  MoveL (T18222) to (121.46, 121.46, 19.3) mm, rotated rx 180 ry 0 rz -180 deg; joints [1.832, 70.767, -37.025, 3.296, -33.786, -2.741]
  Call Extruder 0.54596
  MoveL (T18223) to (103.54, 121.46, 19.3) mm, rotated rx 180 ry 0 rz -180 deg; joints [1.832, 70.767, -37.025, 3.296, -33.786, -2.741]
  Call Extruder 0.54596
  MoveL (T18224) to (103.54, 103.54, 19.3) mm, rotated rx 180 ry 0 rz -180 deg; joints [1.834, 70.589, -36.69, 3.286, -33.943, -2.727]
  Call Extruder 0.02254
  MoveL (T18225) to (104.28, 103.54, 19.3) mm, rotated rx 180 ry 0 rz -180 deg; joints [2.112, 69.848, -35.298, 3.72, -34.607, -3.063]
  Set speed (150.0 mm/s)
  MoveL (T18226) to (103.53, 103.13, 19.3) mm, rotated rx 180 ry 0 rz -180 deg; joints [2.112, 69.848, -35.298, 3.72, -34.607, -3.063]
  Set speed (40.0 mm/s)
  MoveL (T18227) to (103.53, 103.13, 19.3) mm, rotated rx 180 ry 0 rz -180 deg; joints [2.112, 69.848, -35.298, 3.72, -34.607, -3.063]
  Call Extruder 0.55858
  MoveL (T18228) to (121.87, 103.13, 19.3) mm, rotated rx 180 ry 0 rz -180 deg; joints [2.053, 69.842, -35.286, 3.617, -34.609, -2.978]
  Call Extruder 0.57077
  MoveL (T18229) to (121.87, 121.87, 19.3) mm, rotated rx 180 ry 0 rz -180 deg; joints [2.048, 69.847, -35.297, 3.608, -34.604, -2.971]
  Call Extruder 0.57077
  MoveL (T18230) to (103.13, 121.87, 19.3) mm, rotated rx 180 ry 0 rz -180 deg; joints [2.048, 69.847, -35.297, 3.608, -34.604, -2.971]
  Call Extruder 0.57077
  MoveL (T18231) to (103.13, 103.13, 19.3) mm, rotated rx 180 ry 0 rz -180 deg; joints [2.048, 69.847, -35.297, 3.608, -34.604, -2.971]
  Call Extruder 0.01036
  MoveL (T18232) to (103.47, 103.13, 19.3) mm, rotated rx 180 ry 0 rz -180 deg; joints [1.816, 70.466, -36.459, 3.245, -34.05, -2.69]
  Set speed (150.0 mm/s)
  MoveL (T18233) to (102.72, 102.81, 19.3) mm, rotated rx 180 ry 0 rz -180 deg; joints [1.816, 70.466, -36.459, 3.245, -34.05, -2.69]
  Set speed (25.0 mm/s)
  MoveL (T18234) to (102.72, 102.81, 19.3) mm, rotated rx 180 ry 0 rz -180 deg; joints [1.816, 70.466, -36.459, 3.245, -34.05, -2.69]
  Call Extruder 0.00259
  MoveL (T18235) to (102.72, 102.72, 19.3) mm, rotated rx 180 ry 0 rz -180 deg; joints [1.835, 70.04, -35.659, 3.248, -34.424, -2.68]
  Call Extruder 0.59557
  MoveL (T18236) to (122.28, 102.72, 19.3) mm, rotated rx 180 ry 0 rz -180 deg; joints [1.835, 70.04, -35.659, 3.248, -34.424, -2.68]
  Call Extruder 0.59557
  MoveL (T18237) to (122.28, 122.28, 19.3) mm, rotated rx 180 ry 0 rz -180 deg; joints [1.835, 70.04, -35.659, 3.248, -34.424, -2.68]
  Call Extruder 0.59557
  MoveL (T18238) to (102.72, 122.28, 19.3) mm, rotated rx 180 ry 0 rz -180 deg; joints [1.835, 70.04, -35.659, 3.248, -34.424, -2.68]
  Call Extruder 0.59115
  MoveL (T18239) to (102.72, 102.87, 19.3) mm, rotated rx 180 ry 0 rz -180 deg; joints [1.835, 70.04, -35.659, 3.248, -34.424, -2.68]
  Set speed (150.0 mm/s)
  MoveL (T18240) to (102.78, 102.75, 19.3) mm, rotated rx 180 ry 0 rz -180 deg; joints [1.835, 70.04, -35.659, 3.248, -34.424, -2.68]
  Set speed (45.0 mm/s)
  Call Extruder -1.6
  MoveL (T18241) to (102.78, 102.75, 19.3) mm, rotated rx 180 ry 0 rz -180 deg; joints [1.603, 70.67, -36.843, 2.878, -33.861, -2.39]
  Set speed (120.0 mm/s)
  MoveL (T18242) to (102.78, 102.75, 19.3) mm, rotated rx 180 ry 0 rz -180 deg; joints [1.603, 70.67, -36.843, 2.878, -33.861, -2.39]
  Call Extruder -0.05166
  MoveL (T18243) to (102.72, 102.72, 19.3) mm, rotated rx 180 ry 0 rz -180 deg; joints [1.599, 70.675, -36.851, 2.871, -33.857, -2.385]
  Call Extruder -0.32834
  MoveL (T18244) to (103.65, 102.72, 19.3) mm, rotated rx 180 ry 0 rz -180 deg; joints [1.599, 70.675, -36.851, 2.871, -33.857, -2.385]
  Set speed (45.0 mm/s)
  Call Extruder -0.02
  MoveL (T18245) to (103.65, 102.72, 19.3) mm, rotated rx 180 ry 0 rz -180 deg; joints [1.599, 70.675, -36.851, 2.871, -33.857, -2.385]
  Set speed (150.0 mm/s)
  MoveL (T18246) to (103.65, 102.72, 21.3) mm, rotated rx 180 ry 0 rz -180 deg; joints [1.599, 70.675, -36.851, 2.871, -33.857, -2.385]
  MoveL (T18247) to (121.34, 120.51, 21.3) mm, rotated rx 180 ry 0 rz -180 deg; joints [1.539, 70.67, -36.842, 2.763, -33.859, -2.295]
  MoveL (T18248) to (121.34, 120.51, 19.3) mm, rotated rx 180 ry 0 rz -180 deg; joints [1.539, 70.67, -36.842, 2.763, -33.859, -2.295]
  Set speed (40.0 mm/s)
  Call Extruder 2.0
  MoveL (T18249) to (121.34, 120.51, 19.3) mm, rotated rx 180 ry 0 rz -180 deg; joints [1.817, 69.916, -35.425, 3.207, -34.532, -2.643]
  Call Extruder 0.02815
  MoveL (T18250) to (120.69, 121.16, 19.3) mm, rotated rx 180 ry 0 rz -180 deg; joints [1.817, 69.916, -35.425, 3.207, -34.532, -2.643]
  Call Extruder 0.01786
  MoveL (T18251) to (120.11, 121.16, 19.3) mm, rotated rx 180 ry 0 rz -180 deg; joints [1.817, 69.916, -35.425, 3.207, -34.532, -2.643]
  Call Extruder 0.04544
  MoveL (T18252) to (121.16, 120.11, 19.3) mm, rotated rx 180 ry 0 rz -180 deg; joints [1.819, 69.74, -35.095, 3.198, -34.687, -2.631]
  Call Extruder 0.01786
  MoveL (T18253) to (121.16, 119.53, 19.3) mm, rotated rx 180 ry 0 rz -180 deg; joints [1.819, 69.74, -35.095, 3.198, -34.687, -2.631]
  Call Extruder 0.0707
  MoveL (T18254) to (119.53, 121.16, 19.3) mm, rotated rx 180 ry 0 rz -180 deg; joints [1.819, 69.74, -35.095, 3.198, -34.687, -2.631]
  Call Extruder 0.01786
  MoveL (T18255) to (118.95, 121.16, 19.3) mm, rotated rx 180 ry 0 rz -180 deg; joints [1.477, 70.665, -36.833, 2.651, -33.861, -2.202]
  Call Extruder 0.09595
  MoveL (T18256) to (121.16, 118.95, 19.3) mm, rotated rx 180 ry 0 rz -180 deg; joints [1.477, 70.665, -36.833, 2.651, -33.861, -2.202]
  Call Extruder 0.01786
  MoveL (T18257) to (121.16, 118.37, 19.3) mm, rotated rx 180 ry 0 rz -180 deg; joints [1.477, 70.665, -36.833, 2.651, -33.861, -2.202]
  Call Extruder 0.12121
  MoveL (T18258) to (118.37, 121.16, 19.3) mm, rotated rx 180 ry 0 rz -180 deg; joints [1.414, 70.661, -36.825, 2.539, -33.862, -2.108]
  Call Extruder 0.01786
  MoveL (T18259) to (117.79, 121.16, 19.3) mm, rotated rx 180 ry 0 rz -180 deg; joints [1.414, 70.661, -36.825, 2.539, -33.862, -2.108]
  Call Extruder 0.14646
  MoveL (T18260) to (121.16, 117.79, 19.3) mm, rotated rx 180 ry 0 rz -180 deg; joints [1.821, 69.565, -34.766, 3.189, -34.84, -2.618]
  Call Extruder 0.01786
  MoveL (T18261) to (121.16, 117.21, 19.3) mm, rotated rx 180 ry 0 rz -180 deg; joints [1.821, 69.565, -34.766, 3.189, -34.84, -2.618]
  Call Extruder 0.17172
  MoveL (T18262) to (117.21, 121.16, 19.3) mm, rotated rx 180 ry 0 rz -180 deg; joints [1.823, 69.392, -34.441, 3.181, -34.993, -2.607]
  Call Extruder 0.01786
  MoveL (T18263) to (116.62, 121.16, 19.3) mm, rotated rx 180 ry 0 rz -180 deg; joints [1.823, 69.392, -34.441, 3.181, -34.993, -2.607]
  Call Extruder 0.19697
  MoveL (T18264) to (121.16, 116.62, 19.3) mm, rotated rx 180 ry 0 rz -180 deg; joints [1.823, 69.392, -34.441, 3.181, -34.993, -2.607]
  Call Extruder 0.01786
  MoveL (T18265) to (121.16, 116.04, 19.3) mm, rotated rx 180 ry 0 rz -180 deg; joints [1.4, 70.522, -36.565, 2.505, -33.983, -2.078]
  Call Extruder 0.1471
  MoveL (T18266) to (117.77, 119.43, 19.3) mm, rotated rx 180 ry 0 rz -180 deg; joints [1.4, 70.522, -36.565, 2.505, -33.983, -2.078]
  Call Extruder 0.01786
  MoveL (T18267) to (117.77, 118.85, 19.3) mm, rotated rx 180 ry 0 rz -180 deg; joints [1.401, 70.341, -36.225, 2.497, -34.142, -2.067]
  Call Extruder 0.1471
  MoveL (T18268) to (121.16, 115.46, 19.3) mm, rotated rx 180 ry 0 rz -180 deg; joints [1.401, 70.341, -36.225, 2.497, -34.142, -2.067]
  Call Extruder 0.01786
  MoveL (T18269) to (121.16, 114.88, 19.3) mm, rotated rx 180 ry 0 rz -180 deg; joints [1.825, 69.219, -34.117, 3.172, -35.144, -2.595]
  Call Extruder 0.1471
  MoveL (T18270) to (117.77, 118.27, 19.3) mm, rotated rx 180 ry 0 rz -180 deg; joints [1.825, 69.219, -34.117, 3.172, -35.144, -2.595]
  Call Extruder 0.0059
  MoveL (T18271) to (117.77, 118.07, 19.3) mm, rotated rx 180 ry 0 rz -180 deg; joints [1.827, 69.049, -33.796, 3.164, -35.294, -2.583]
  Call Extruder 0.00889
  MoveL (T18272) to (117.64, 117.82, 19.3) mm, rotated rx 180 ry 0 rz -180 deg; joints [1.827, 69.049, -33.796, 3.164, -35.294, -2.583]
  Call Extruder 0.15283
  MoveL (T18273) to (121.16, 114.3, 19.3) mm, rotated rx 180 ry 0 rz -180 deg; joints [1.827, 69.049, -33.796, 3.164, -35.294, -2.583]
  Call Extruder 0.01786
  MoveL (T18274) to (121.16, 113.72, 19.3) mm, rotated rx 180 ry 0 rz -180 deg; joints [1.403, 70.162, -35.888, 2.49, -34.299, -2.057]
  Call Extruder 0.16138
  MoveL (T18275) to (117.44, 117.43, 19.3) mm, rotated rx 180 ry 0 rz -180 deg; joints [1.403, 70.162, -35.888, 2.49, -34.299, -2.057]
  Call Extruder 0.01327
  MoveL (T18276) to (117.25, 117.05, 19.3) mm, rotated rx 180 ry 0 rz -180 deg; joints [1.404, 69.984, -35.554, 2.483, -34.455, -2.048]
  Call Extruder 0.16993
  MoveL (T18277) to (121.16, 113.14, 19.3) mm, rotated rx 180 ry 0 rz -180 deg; joints [1.404, 69.984, -35.554, 2.483, -34.455, -2.048]
  Call Extruder 0.01786
  MoveL (T18278) to (121.16, 112.56, 19.3) mm, rotated rx 180 ry 0 rz -180 deg; joints [1.404, 69.984, -35.554, 2.483, -34.455, -2.048]
  Call Extruder 0.17848
  MoveL (T18279) to (117.05, 116.66, 19.3) mm, rotated rx 180 ry 0 rz -180 deg; joints [1.829, 68.879, -33.477, 3.156, -35.443, -2.572]
  Call Extruder 0.01327
  MoveL (T18280) to (116.85, 116.28, 19.3) mm, rotated rx 180 ry 0 rz -180 deg; joints [1.829, 68.879, -33.477, 3.156, -35.443, -2.572]
  Call Extruder 0.18703
  MoveL (T18281) to (121.16, 111.98, 19.3) mm, rotated rx 180 ry 0 rz -180 deg; joints [1.829, 68.879, -33.477, 3.156, -35.443, -2.572]
  Call Extruder 0.01786
  MoveL (T18282) to (121.16, 111.4, 19.3) mm, rotated rx 180 ry 0 rz -180 deg; joints [1.831, 68.775, -33.283, 3.151, -35.534, -2.565]
  Call Extruder 0.19558
  MoveL (T18283) to (116.66, 115.89, 19.3) mm, rotated rx 180 ry 0 rz -180 deg; joints [1.831, 68.775, -33.283, 3.151, -35.534, -2.565]
  Call Extruder 0.01327
  MoveL (T18284) to (116.46, 115.51, 19.3) mm, rotated rx 180 ry 0 rz -180 deg; joints [1.831, 68.775, -33.283, 3.151, -35.534, -2.565]
  Call Extruder 0.20412
  MoveL (T18285) to (121.16, 110.81, 19.3) mm, rotated rx 180 ry 0 rz -180 deg; joints [1.831, 68.775, -33.283, 3.151, -35.534, -2.565]
  Call Extruder 0.01786
  MoveL (T18286) to (121.16, 110.23, 19.3) mm, rotated rx 180 ry 0 rz -180 deg; joints [1.828, 68.761, -33.255, 3.146, -35.546, -2.561]
  Call Extruder 0.21267
  MoveL (T18287) to (116.26, 115.13, 19.3) mm, rotated rx 180 ry 0 rz -180 deg; joints [1.828, 68.761, -33.255, 3.146, -35.546, -2.561]
  Call Extruder 0.01327
  MoveL (T18288) to (116.07, 114.74, 19.3) mm, rotated rx 180 ry 0 rz -180 deg; joints [1.828, 68.761, -33.255, 3.146, -35.546, -2.561]
  Call Extruder 0.22122
  MoveL (T18289) to (121.16, 109.65, 19.3) mm, rotated rx 180 ry 0 rz -180 deg; joints [1.82, 68.738, -33.212, 3.131, -35.566, -2.548]
  Call Extruder 0.01786
  MoveL (T18290) to (121.16, 109.07, 19.3) mm, rotated rx 180 ry 0 rz -180 deg; joints [1.82, 68.738, -33.212, 3.131, -35.566, -2.548]
  Call Extruder 0.22977
  MoveL (T18291) to (115.87, 114.36, 19.3) mm, rotated rx 180 ry 0 rz -180 deg; joints [1.406, 69.808, -35.222, 2.476, -34.611, -2.038]
  Call Extruder 0.01327
  MoveL (T18292) to (115.67, 113.97, 19.3) mm, rotated rx 180 ry 0 rz -180 deg; joints [1.406, 69.808, -35.222, 2.476, -34.611, -2.038]
  Call Extruder 0.23832
  MoveL (T18293) to (121.16, 108.49, 19.3) mm, rotated rx 180 ry 0 rz -180 deg; joints [1.408, 69.632, -34.893, 2.469, -34.765, -2.029]
  Call Extruder 0.01786
  MoveL (T18294) to (121.16, 107.91, 19.3) mm, rotated rx 180 ry 0 rz -180 deg; joints [1.408, 69.632, -34.893, 2.469, -34.765, -2.029]
  Call Extruder 0.24687
  MoveL (T18295) to (115.48, 113.59, 19.3) mm, rotated rx 180 ry 0 rz -180 deg; joints [1.408, 69.632, -34.893, 2.469, -34.765, -2.029]
  Call Extruder 0.01327
  MoveL (T18296) to (115.28, 113.2, 19.3) mm, rotated rx 180 ry 0 rz -180 deg; joints [1.79, 68.651, -33.049, 3.072, -35.641, -2.498]
  Call Extruder 0.25542
  MoveL (T18297) to (121.16, 107.33, 19.3) mm, rotated rx 180 ry 0 rz -180 deg; joints [1.79, 68.651, -33.049, 3.072, -35.641, -2.498]
  Call Extruder 0.01786
  MoveL (T18298) to (121.16, 106.75, 19.3) mm, rotated rx 180 ry 0 rz -180 deg; joints [1.79, 68.651, -33.049, 3.072, -35.641, -2.498]
  Call Extruder 0.26397
  MoveL (T18299) to (115.08, 112.82, 19.3) mm, rotated rx 180 ry 0 rz -180 deg; joints [1.759, 68.565, -32.887, 3.014, -35.715, -2.448]
  Call Extruder 0.01327
  MoveL (T18300) to (114.89, 112.44, 19.3) mm, rotated rx 180 ry 0 rz -180 deg; joints [1.759, 68.565, -32.887, 3.014, -35.715, -2.448]
  Call Extruder 0.27252
  MoveL (T18301) to (121.16, 106.17, 19.3) mm, rotated rx 180 ry 0 rz -180 deg; joints [1.759, 68.565, -32.887, 3.014, -35.715, -2.448]
  Call Extruder 0.01786
  MoveL (T18302) to (121.16, 105.59, 19.3) mm, rotated rx 180 ry 0 rz -180 deg; joints [1.409, 69.458, -34.566, 2.462, -34.917, -2.019]
  Call Extruder 0.13907
  MoveL (T18303) to (117.96, 108.79, 19.3) mm, rotated rx 180 ry 0 rz -180 deg; joints [1.409, 69.458, -34.566, 2.462, -34.917, -2.019]
  Call Extruder 0.01777
  MoveL (T18304) to (117.96, 109.36, 19.3) mm, rotated rx 180 ry 0 rz -180 deg; joints [1.409, 69.458, -34.566, 2.462, -34.917, -2.019]
  Call Extruder 0.01777
  MoveL (T18305) to (117.38, 109.36, 19.3) mm, rotated rx 180 ry 0 rz -180 deg; joints [1.411, 69.286, -34.241, 2.456, -35.069, -2.01]
  Call Extruder 0.11687
  MoveL (T18306) to (114.69, 112.05, 19.3) mm, rotated rx 180 ry 0 rz -180 deg; joints [1.411, 69.286, -34.241, 2.456, -35.069, -2.01]
  Call Extruder 0.01327
  MoveL (T18307) to (114.49, 111.67, 19.3) mm, rotated rx 180 ry 0 rz -180 deg; joints [1.728, 68.479, -32.726, 2.956, -35.789, -2.399]
  Call Extruder 0.10016
  MoveL (T18308) to (116.8, 109.36, 19.3) mm, rotated rx 180 ry 0 rz -180 deg; joints [1.728, 68.479, -32.726, 2.956, -35.789, -2.399]
  Call Extruder 0.01786
  MoveL (T18309) to (116.22, 109.36, 19.3) mm, rotated rx 180 ry 0 rz -180 deg; joints [1.698, 68.393, -32.565, 2.899, -35.863, -2.35]
  Call Extruder 0.08346
  MoveL (T18310) to (114.3, 111.28, 19.3) mm, rotated rx 180 ry 0 rz -180 deg; joints [1.698, 68.393, -32.565, 2.899, -35.863, -2.35]
  Call Extruder 0.01327
  MoveL (T18311) to (114.1, 110.9, 19.3) mm, rotated rx 180 ry 0 rz -180 deg; joints [1.698, 68.393, -32.565, 2.899, -35.863, -2.35]
  Call Extruder 0.06675
  MoveL (T18312) to (115.64, 109.36, 19.3) mm, rotated rx 180 ry 0 rz -180 deg; joints [1.698, 68.393, -32.565, 2.899, -35.863, -2.35]
  Call Extruder 0.01786
  MoveL (T18313) to (115.06, 109.36, 19.3) mm, rotated rx 180 ry 0 rz -180 deg; joints [1.412, 69.114, -33.919, 2.449, -35.22, -2.001]
  Call Extruder 0.05004
  MoveL (T18314) to (113.9, 110.52, 19.3) mm, rotated rx 180 ry 0 rz -180 deg; joints [1.412, 69.114, -33.919, 2.449, -35.22, -2.001]
  Call Extruder 0.01327
  MoveL (T18315) to (113.71, 110.13, 19.3) mm, rotated rx 180 ry 0 rz -180 deg; joints [1.412, 69.114, -33.919, 2.449, -35.22, -2.001]
  Call Extruder 0.03334
  MoveL (T18316) to (114.47, 109.36, 19.3) mm, rotated rx 180 ry 0 rz -180 deg; joints [1.414, 68.944, -33.599, 2.443, -35.369, -1.992]
  Call Extruder 0.01786
  MoveL (T18317) to (113.89, 109.36, 19.3) mm, rotated rx 180 ry 0 rz -180 deg; joints [1.414, 68.944, -33.599, 2.443, -35.369, -1.992]
  Call Extruder 0.02255
  MoveL (T18318) to (113.37, 109.88, 19.3) mm, rotated rx 180 ry 0 rz -180 deg; joints [1.842, 67.884, -31.608, 3.11, -36.316, -2.507]
  Set speed (45.0 mm/s)
  Call Extruder -1.6
  MoveL (T18319) to (113.37, 109.88, 19.3) mm, rotated rx 180 ry 0 rz -180 deg; joints [1.842, 67.884, -31.608, 3.11, -36.316, -2.507]
  Set speed (120.0 mm/s)
  MoveL (T18320) to (113.37, 109.88, 19.3) mm, rotated rx 180 ry 0 rz -180 deg; joints [1.844, 67.721, -31.303, 3.103, -36.458, -2.497]
  Call Extruder -0.26134
  MoveL (T18321) to (113.89, 109.36, 19.3) mm, rotated rx 180 ry 0 rz -180 deg; joints [1.844, 67.721, -31.303, 3.103, -36.458, -2.497]
  Call Extruder -0.11866
  MoveL (T18322) to (114.23, 109.36, 19.3) mm, rotated rx 180 ry 0 rz -180 deg; joints [1.415, 68.775, -33.282, 2.437, -35.517, -1.984]
  Set speed (45.0 mm/s)
  Call Extruder -0.02
  MoveL (T18323) to (114.23, 109.36, 19.3) mm, rotated rx 180 ry 0 rz -180 deg; joints [1.417, 68.607, -32.966, 2.431, -35.665, -1.975]
  Set speed (150.0 mm/s)
  MoveL (T18324) to (114.23, 109.36, 21.3) mm, rotated rx 180 ry 0 rz -180 deg; joints [1.417, 68.607, -32.966, 2.431, -35.665, -1.975]
  MoveL (T18325) to (117.77, 108.39, 21.3) mm, rotated rx 180 ry 0 rz -180 deg; joints [1.846, 67.561, -31.001, 3.097, -36.599, -2.487]
  MoveL (T18326) to (117.77, 108.39, 19.3) mm, rotated rx 180 ry 0 rz -180 deg; joints [1.846, 67.561, -31.001, 3.097, -36.599, -2.487]
  Set speed (40.0 mm/s)
  Call Extruder 2.0
  MoveL (T18327) to (117.77, 108.39, 19.3) mm, rotated rx 180 ry 0 rz -180 deg; joints [1.846, 67.561, -31.001, 3.097, -36.599, -2.487]
  Call Extruder 0.14703
  MoveL (T18328) to (121.16, 105.01, 19.3) mm, rotated rx 180 ry 0 rz -180 deg; joints [1.848, 67.401, -30.701, 3.09, -36.74, -2.477]
  Call Extruder 0.01786
  MoveL (T18329) to (121.16, 104.42, 19.3) mm, rotated rx 180 ry 0 rz -180 deg; joints [1.848, 67.401, -30.701, 3.09, -36.74, -2.477]
  Call Extruder 0.13907
  MoveL (T18330) to (117.96, 107.62, 19.3) mm, rotated rx 180 ry 0 rz -180 deg; joints [1.848, 67.401, -30.701, 3.09, -36.74, -2.477]
  Call Extruder 0.01786
  MoveL (T18331) to (117.96, 107.04, 19.3) mm, rotated rx 180 ry 0 rz -180 deg; joints [1.418, 68.44, -32.653, 2.425, -35.811, -1.967]
  Call Extruder 0.13906
  MoveL (T18332) to (121.16, 103.84, 19.3) mm, rotated rx 180 ry 0 rz -180 deg; joints [1.418, 68.44, -32.653, 2.425, -35.811, -1.967]
  Call Extruder 0.01786
  MoveL (T18333) to (120.58, 103.84, 19.3) mm, rotated rx 180 ry 0 rz -180 deg; joints [1.42, 68.274, -32.342, 2.419, -35.957, -1.958]
  Call Extruder 0.11381
  MoveL (T18334) to (117.96, 106.46, 19.3) mm, rotated rx 180 ry 0 rz -180 deg; joints [1.42, 68.274, -32.342, 2.419, -35.957, -1.958]
  Call Extruder 0.01786
  MoveL (T18335) to (117.96, 105.88, 19.3) mm, rotated rx 180 ry 0 rz -180 deg; joints [1.42, 68.274, -32.342, 2.419, -35.957, -1.958]
  Call Extruder 0.08856
  MoveL (T18336) to (119.99, 103.84, 19.3) mm, rotated rx 180 ry 0 rz -180 deg; joints [1.85, 67.241, -30.402, 3.083, -36.879, -2.467]
  Call Extruder 0.01786
  MoveL (T18337) to (119.41, 103.84, 19.3) mm, rotated rx 180 ry 0 rz -180 deg; joints [1.85, 67.241, -30.402, 3.083, -36.879, -2.467]
  Call Extruder 0.0633
  MoveL (T18338) to (117.96, 105.3, 19.3) mm, rotated rx 180 ry 0 rz -180 deg; joints [1.85, 67.241, -30.402, 3.083, -36.879, -2.467]
  Call Extruder 0.00424
  MoveL (T18339) to (117.96, 105.16, 19.3) mm, rotated rx 180 ry 0 rz -180 deg; joints [1.852, 67.083, -30.105, 3.077, -37.018, -2.457]
  Call Extruder 0.01362
  MoveL (T18340) to (117.51, 105.16, 19.3) mm, rotated rx 180 ry 0 rz -180 deg; joints [1.422, 68.11, -32.033, 2.413, -36.101, -1.95]
  Call Extruder 0.0573
  MoveL (T18341) to (118.83, 103.84, 19.3) mm, rotated rx 180 ry 0 rz -180 deg; joints [1.422, 68.11, -32.033, 2.413, -36.101, -1.95]
  Call Extruder 0.01786
  MoveL (T18342) to (118.25, 103.84, 19.3) mm, rotated rx 180 ry 0 rz -180 deg; joints [1.422, 68.11, -32.033, 2.413, -36.101, -1.95]
  Call Extruder 0.0573
  MoveL (T18343) to (116.93, 105.16, 19.3) mm, rotated rx 180 ry 0 rz -180 deg; joints [1.422, 68.11, -32.033, 2.413, -36.101, -1.95]
  Call Extruder 0.01786
  MoveL (T18344) to (116.35, 105.16, 19.3) mm, rotated rx 180 ry 0 rz -180 deg; joints [1.423, 67.946, -31.725, 2.407, -36.245, -1.942]
  Call Extruder 0.0573
  MoveL (T18345) to (117.67, 103.84, 19.3) mm, rotated rx 180 ry 0 rz -180 deg; joints [1.423, 67.946, -31.725, 2.407, -36.245, -1.942]
  Call Extruder 0.01786
  MoveL (T18346) to (117.09, 103.84, 19.3) mm, rotated rx 180 ry 0 rz -180 deg; joints [1.423, 67.946, -31.725, 2.407, -36.245, -1.942]
  Call Extruder 0.0573
  MoveL (T18347) to (115.77, 105.16, 19.3) mm, rotated rx 180 ry 0 rz -180 deg; joints [1.423, 67.946, -31.725, 2.407, -36.245, -1.942]
  Call Extruder 0.01786
  MoveL (T18348) to (115.19, 105.16, 19.3) mm, rotated rx 180 ry 0 rz -180 deg; joints [1.854, 66.926, -29.809, 3.07, -37.156, -2.448]
  Call Extruder 0.0573
  MoveL (T18349) to (116.51, 103.84, 19.3) mm, rotated rx 180 ry 0 rz -180 deg; joints [1.854, 66.926, -29.809, 3.07, -37.156, -2.448]
  Call Extruder 0.01786
  MoveL (T18350) to (115.93, 103.84, 19.3) mm, rotated rx 180 ry 0 rz -180 deg; joints [1.856, 66.77, -29.516, 3.064, -37.293, -2.438]
  Call Extruder 0.0573
  MoveL (T18351) to (114.61, 105.16, 19.3) mm, rotated rx 180 ry 0 rz -180 deg; joints [1.856, 66.77, -29.516, 3.064, -37.293, -2.438]
  Call Extruder 0.01786
  MoveL (T18352) to (114.03, 105.16, 19.3) mm, rotated rx 180 ry 0 rz -180 deg; joints [1.856, 66.77, -29.516, 3.064, -37.293, -2.438]
  Call Extruder 0.0573
  MoveL (T18353) to (115.35, 103.84, 19.3) mm, rotated rx 180 ry 0 rz -180 deg; joints [1.425, 67.784, -31.42, 2.402, -36.388, -1.934]
  Call Extruder 0.01786
  MoveL (T18354) to (114.77, 103.84, 19.3) mm, rotated rx 180 ry 0 rz -180 deg; joints [1.425, 67.784, -31.42, 2.402, -36.388, -1.934]
  Call Extruder 0.0573
  MoveL (T18355) to (113.45, 105.16, 19.3) mm, rotated rx 180 ry 0 rz -180 deg; joints [1.426, 67.622, -31.117, 2.397, -36.529, -1.926]
  Call Extruder 0.01786
  MoveL (T18356) to (112.87, 105.16, 19.3) mm, rotated rx 180 ry 0 rz -180 deg; joints [1.426, 67.622, -31.117, 2.397, -36.529, -1.926]
  Call Extruder 0.0573
  MoveL (T18357) to (114.18, 103.84, 19.3) mm, rotated rx 180 ry 0 rz -180 deg; joints [1.827, 66.685, -29.358, 3.011, -37.366, -2.394]
  Call Extruder 0.01786
  MoveL (T18358) to (113.6, 103.84, 19.3) mm, rotated rx 180 ry 0 rz -180 deg; joints [1.827, 66.685, -29.358, 3.011, -37.366, -2.394]
  Call Extruder 0.0573
  MoveL (T18359) to (112.28, 105.16, 19.3) mm, rotated rx 180 ry 0 rz -180 deg; joints [1.827, 66.685, -29.358, 3.011, -37.366, -2.394]
  Call Extruder 0.01786
  MoveL (T18360) to (111.7, 105.16, 19.3) mm, rotated rx 180 ry 0 rz -180 deg; joints [1.796, 66.605, -29.207, 2.955, -37.435, -2.347]
  Call Extruder 0.0573
  MoveL (T18361) to (113.02, 103.84, 19.3) mm, rotated rx 180 ry 0 rz -180 deg; joints [1.796, 66.605, -29.207, 2.955, -37.435, -2.347]
  Call Extruder 0.01786
  MoveL (T18362) to (112.44, 103.84, 19.3) mm, rotated rx 180 ry 0 rz -180 deg; joints [1.796, 66.605, -29.207, 2.955, -37.435, -2.347]
  Call Extruder 0.0573
  MoveL (T18363) to (111.12, 105.16, 19.3) mm, rotated rx 180 ry 0 rz -180 deg; joints [1.796, 66.605, -29.207, 2.955, -37.435, -2.347]
  Call Extruder 0.01786
  MoveL (T18364) to (110.54, 105.16, 19.3) mm, rotated rx 180 ry 0 rz -180 deg; joints [1.428, 67.462, -30.815, 2.391, -36.67, -1.918]
  Call Extruder 0.0573
  MoveL (T18365) to (111.86, 103.84, 19.3) mm, rotated rx 180 ry 0 rz -180 deg; joints [1.428, 67.462, -30.815, 2.391, -36.67, -1.918]
  Call Extruder 0.01786
  MoveL (T18366) to (111.28, 103.84, 19.3) mm, rotated rx 180 ry 0 rz -180 deg; joints [1.428, 67.462, -30.815, 2.391, -36.67, -1.918]
  Call Extruder 0.0573
  MoveL (T18367) to (109.96, 105.16, 19.3) mm, rotated rx 180 ry 0 rz -180 deg; joints [1.429, 67.302, -30.516, 2.386, -36.81, -1.911]
  Call Extruder 0.01786
  MoveL (T18368) to (109.38, 105.16, 19.3) mm, rotated rx 180 ry 0 rz -180 deg; joints [1.429, 67.302, -30.516, 2.386, -36.81, -1.911]
  Call Extruder 0.0573
  MoveL (T18369) to (110.7, 103.84, 19.3) mm, rotated rx 180 ry 0 rz -180 deg; joints [1.429, 67.302, -30.516, 2.386, -36.81, -1.911]
  Call Extruder 0.01786
  MoveL (T18370) to (110.12, 103.84, 19.3) mm, rotated rx 180 ry 0 rz -180 deg; joints [1.765, 66.525, -29.057, 2.899, -37.503, -2.301]
  Call Extruder 0.0573
  MoveL (T18371) to (108.8, 105.16, 19.3) mm, rotated rx 180 ry 0 rz -180 deg; joints [1.765, 66.525, -29.057, 2.899, -37.503, -2.301]
  Call Extruder 0.01786
  MoveL (T18372) to (108.22, 105.16, 19.3) mm, rotated rx 180 ry 0 rz -180 deg; joints [1.765, 66.525, -29.057, 2.899, -37.503, -2.301]
  Call Extruder 0.06527
  MoveL (T18373) to (109.72, 103.66, 19.3) mm, rotated rx 180 ry 0 rz -180 deg; joints [1.734, 66.446, -28.908, 2.844, -37.572, -2.255]
  Set speed (45.0 mm/s)
  Call Extruder -1.6
  MoveL (T18374) to (109.72, 103.66, 19.3) mm, rotated rx 180 ry 0 rz -180 deg; joints [1.734, 66.446, -28.908, 2.844, -37.572, -2.255]
  Set speed (120.0 mm/s)
  MoveL (T18375) to (109.72, 103.66, 19.3) mm, rotated rx 180 ry 0 rz -180 deg; joints [1.734, 66.446, -28.908, 2.844, -37.572, -2.255]
  Call Extruder -0.38
  MoveL (T18376) to (108.97, 104.42, 19.3) mm, rotated rx 180 ry 0 rz -180 deg; joints [1.431, 67.143, -30.218, 2.381, -36.949, -1.903]
  Set speed (45.0 mm/s)
  Call Extruder -0.02
  MoveL (T18377) to (108.97, 104.42, 19.3) mm, rotated rx 180 ry 0 rz -180 deg; joints [1.431, 67.143, -30.218, 2.381, -36.949, -1.903]
  Set speed (150.0 mm/s)
  MoveL (T18378) to (108.97, 104.42, 21.3) mm, rotated rx 180 ry 0 rz -180 deg; joints [1.431, 67.143, -30.218, 2.381, -36.949, -1.903]
  MoveL (T18379) to (111.87, 115.45, 21.3) mm, rotated rx 180 ry 0 rz -180 deg; joints [1.433, 66.986, -29.922, 2.376, -37.087, -1.896]
  MoveL (T18380) to (111.87, 115.45, 19.3) mm, rotated rx 180 ry 0 rz -180 deg; joints [1.433, 66.986, -29.922, 2.376, -37.087, -1.896]
  Set speed (40.0 mm/s)
  Call Extruder 2.0
  MoveL (T18381) to (111.87, 115.45, 19.3) mm, rotated rx 180 ry 0 rz -180 deg; joints [1.433, 66.986, -29.922, 2.376, -37.087, -1.896]
  Call Extruder 0.022
  MoveL (T18382) to (111.36, 115.96, 19.3) mm, rotated rx 180 ry 0 rz -180 deg; joints [1.433, 66.986, -29.922, 2.376, -37.087, -1.896]
  Call Extruder 0.01786
  MoveL (T18383) to (110.78, 115.96, 19.3) mm, rotated rx 180 ry 0 rz -180 deg; joints [1.702, 66.367, -28.76, 2.788, -37.64, -2.209]
  Call Extruder 0.03281
  MoveL (T18384) to (111.54, 115.21, 19.3) mm, rotated rx 180 ry 0 rz -180 deg; joints [1.702, 66.367, -28.76, 2.788, -37.64, -2.209]
  Call Extruder 0.01328
  MoveL (T18385) to (111.34, 114.82, 19.3) mm, rotated rx 180 ry 0 rz -180 deg; joints [1.702, 66.367, -28.76, 2.788, -37.64, -2.209]
  Call Extruder 0.04953
  MoveL (T18386) to (110.2, 115.96, 19.3) mm, rotated rx 180 ry 0 rz -180 deg; joints [1.671, 66.288, -28.611, 2.733, -37.708, -2.163]
  Call Extruder 0.01786
  MoveL (T18387) to (109.62, 115.96, 19.3) mm, rotated rx 180 ry 0 rz -180 deg; joints [1.671, 66.288, -28.611, 2.733, -37.708, -2.163]
  Call Extruder 0.06625
  MoveL (T18388) to (111.14, 114.44, 19.3) mm, rotated rx 180 ry 0 rz -180 deg; joints [1.434, 66.829, -29.628, 2.371, -37.225, -1.889]
  Call Extruder 0.01328
  MoveL (T18389) to (110.95, 114.05, 19.3) mm, rotated rx 180 ry 0 rz -180 deg; joints [1.434, 66.829, -29.628, 2.371, -37.225, -1.889]
  Call Extruder 0.08298
  MoveL (T18390) to (109.04, 115.96, 19.3) mm, rotated rx 180 ry 0 rz -180 deg; joints [1.436, 66.673, -29.335, 2.367, -37.362, -1.881]
  Call Extruder 0.01786
  MoveL (T18391) to (108.46, 115.96, 19.3) mm, rotated rx 180 ry 0 rz -180 deg; joints [1.629, 66.233, -28.509, 2.662, -37.754, -2.105]
  Call Extruder 0.10562
  MoveL (T18392) to (110.89, 113.53, 19.3) mm, rotated rx 180 ry 0 rz -180 deg; joints [1.629, 66.233, -28.509, 2.662, -37.754, -2.105]
  Set speed (45.0 mm/s)
  Call Extruder -1.6
  MoveL (T18393) to (110.89, 113.53, 19.3) mm, rotated rx 180 ry 0 rz -180 deg; joints [1.629, 66.233, -28.509, 2.662, -37.754, -2.105]
  Set speed (120.0 mm/s)
  MoveL (T18394) to (110.89, 113.53, 19.3) mm, rotated rx 180 ry 0 rz -180 deg; joints [1.565, 66.229, -28.501, 2.556, -37.755, -2.022]
  Call Extruder -0.38
  MoveL (T18395) to (110.13, 114.29, 19.3) mm, rotated rx 180 ry 0 rz -180 deg; joints [1.565, 66.229, -28.501, 2.556, -37.755, -2.022]
  Set speed (45.0 mm/s)
  Call Extruder -0.02
  MoveL (T18396) to (110.13, 114.29, 19.3) mm, rotated rx 180 ry 0 rz -180 deg; joints [1.565, 66.229, -28.501, 2.556, -37.755, -2.022]
  Set speed (150.0 mm/s)
  MoveL (T18397) to (110.13, 114.29, 21.3) mm, rotated rx 180 ry 0 rz -180 deg; joints [1.565, 66.229, -28.501, 2.556, -37.755, -2.022]
  MoveL (T18398) to (117.22, 119.98, 21.3) mm, rotated rx 180 ry 0 rz -180 deg; joints [1.437, 66.519, -29.045, 2.362, -37.497, -1.874]
  MoveL (T18399) to (117.22, 119.98, 19.3) mm, rotated rx 180 ry 0 rz -180 deg; joints [1.437, 66.519, -29.045, 2.362, -37.497, -1.874]
  Set speed (40.0 mm/s)
  Call Extruder 2.0
  MoveL (T18400) to (117.22, 119.98, 19.3) mm, rotated rx 180 ry 0 rz -180 deg; joints [1.439, 66.364, -28.755, 2.357, -37.633, -1.867]
  Call Extruder 0.05113
  MoveL (T18401) to (116.04, 121.16, 19.3) mm, rotated rx 180 ry 0 rz -180 deg; joints [1.439, 66.364, -28.755, 2.357, -37.633, -1.867]
  Call Extruder 0.01786
  MoveL (T18402) to (115.46, 121.16, 19.3) mm, rotated rx 180 ry 0 rz -180 deg; joints [1.521, 66.179, -28.407, 2.482, -37.798, -1.962]
  Call Extruder 0.04317
  MoveL (T18403) to (116.46, 120.16, 19.3) mm, rotated rx 180 ry 0 rz -180 deg; joints [1.521, 66.179, -28.407, 2.482, -37.798, -1.962]
  Call Extruder 0.01786
  MoveL (T18404) to (115.88, 120.16, 19.3) mm, rotated rx 180 ry 0 rz -180 deg; joints [1.521, 66.179, -28.407, 2.482, -37.798, -1.962]
  Call Extruder 0.04317
  MoveL (T18405) to (114.88, 121.16, 19.3) mm, rotated rx 180 ry 0 rz -180 deg; joints [1.521, 66.179, -28.407, 2.482, -37.798, -1.962]
  Call Extruder 0.01786
  MoveL (T18406) to (114.3, 121.16, 19.3) mm, rotated rx 180 ry 0 rz -180 deg; joints [1.521, 66.179, -28.407, 2.482, -37.798, -1.962]
  Call Extruder 0.04317
  MoveL (T18407) to (115.29, 120.16, 19.3) mm, rotated rx 180 ry 0 rz -180 deg; joints [1.521, 66.179, -28.407, 2.482, -37.798, -1.962]
  Call Extruder 0.01786
  MoveL (T18408) to (114.71, 120.16, 19.3) mm, rotated rx 180 ry 0 rz -180 deg; joints [1.521, 66.179, -28.407, 2.482, -37.798, -1.962]
  Call Extruder 0.04317
  MoveL (T18409) to (113.72, 121.16, 19.3) mm, rotated rx 180 ry 0 rz -180 deg; joints [1.521, 66.179, -28.407, 2.482, -37.798, -1.962]
  Call Extruder 0.01786
  MoveL (T18410) to (113.14, 121.16, 19.3) mm, rotated rx 180 ry 0 rz -180 deg; joints [1.521, 66.179, -28.407, 2.482, -37.798, -1.962]
  Call Extruder 0.04317
  MoveL (T18411) to (114.13, 120.16, 19.3) mm, rotated rx 180 ry 0 rz -180 deg; joints [1.439, 66.364, -28.755, 2.357, -37.633, -1.867]
  Call Extruder 0.01786
  MoveL (T18412) to (113.55, 120.16, 19.3) mm, rotated rx 180 ry 0 rz -180 deg; joints [1.439, 66.364, -28.755, 2.357, -37.633, -1.867]
  Call Extruder 0.04317
  MoveL (T18413) to (112.56, 121.16, 19.3) mm, rotated rx 180 ry 0 rz -180 deg; joints [1.439, 66.37, -28.766, 2.357, -37.627, -1.867]
  Call Extruder 0.01786
  MoveL (T18414) to (111.98, 121.16, 19.3) mm, rotated rx 180 ry 0 rz -180 deg; joints [1.439, 66.37, -28.766, 2.357, -37.627, -1.867]
  Call Extruder 0.04317
  MoveL (T18415) to (112.97, 120.16, 19.3) mm, rotated rx 180 ry 0 rz -180 deg; joints [1.439, 66.37, -28.766, 2.357, -37.627, -1.867]
  Call Extruder 0.01786
  MoveL (T18416) to (112.39, 120.16, 19.3) mm, rotated rx 180 ry 0 rz -180 deg; joints [1.439, 66.37, -28.766, 2.357, -37.627, -1.867]
  Call Extruder 0.04317
  MoveL (T18417) to (111.4, 121.16, 19.3) mm, rotated rx 180 ry 0 rz -180 deg; joints [1.439, 66.37, -28.766, 2.357, -37.627, -1.867]
  Call Extruder 0.01786
  MoveL (T18418) to (110.81, 121.16, 19.3) mm, rotated rx 180 ry 0 rz -180 deg; joints [1.439, 66.37, -28.766, 2.357, -37.627, -1.867]
  Call Extruder 0.04317
  MoveL (T18419) to (111.81, 120.16, 19.3) mm, rotated rx 180 ry 0 rz -180 deg; joints [1.439, 66.37, -28.766, 2.357, -37.627, -1.867]
  Call Extruder 0.01786
  MoveL (T18420) to (111.23, 120.16, 19.3) mm, rotated rx 180 ry 0 rz -180 deg; joints [1.439, 66.37, -28.766, 2.357, -37.627, -1.867]
  Call Extruder 0.04317
  MoveL (T18421) to (110.23, 121.16, 19.3) mm, rotated rx 180 ry 0 rz -180 deg; joints [1.439, 66.135, -28.73, 2.368, -37.428, -1.881]
  Call Extruder 0.01786
  MoveL (T18422) to (109.65, 121.16, 19.3) mm, rotated rx 180 ry 0 rz -180 deg; joints [1.888, 67.7, -31.262, 3.176, -36.479, -2.555]
  Call Extruder 0.04317
  MoveL (T18423) to (110.65, 120.16, 19.3) mm, rotated rx 180 ry 0 rz -180 deg; joints [1.888, 67.7, -31.262, 3.176, -36.479, -2.555]
  Call Extruder 0.01786
  MoveL (T18424) to (110.07, 120.16, 19.3) mm, rotated rx 180 ry 0 rz -180 deg; joints [1.888, 67.7, -31.262, 3.176, -36.479, -2.555]
  Call Extruder 0.04317
  MoveL (T18425) to (109.07, 121.16, 19.3) mm, rotated rx 180 ry 0 rz -180 deg; joints [1.888, 67.7, -31.262, 3.176, -36.479, -2.555]
  Call Extruder 0.01786
  MoveL (T18426) to (108.49, 121.16, 19.3) mm, rotated rx 180 ry 0 rz -180 deg; joints [1.888, 67.7, -31.262, 3.176, -36.479, -2.555]
  Call Extruder 0.04317
  MoveL (T18427) to (109.48, 120.16, 19.3) mm, rotated rx 180 ry 0 rz -180 deg; joints [1.888, 67.7, -31.262, 3.176, -36.479, -2.555]
  Call Extruder 0.01786
  MoveL (T18428) to (108.9, 120.16, 19.3) mm, rotated rx 180 ry 0 rz -180 deg; joints [1.888, 67.7, -31.262, 3.176, -36.479, -2.555]
  Call Extruder 0.04317
  MoveL (T18429) to (107.91, 121.16, 19.3) mm, rotated rx 180 ry 0 rz -180 deg; joints [1.888, 67.7, -31.262, 3.176, -36.479, -2.555]
  Call Extruder 0.01786
  MoveL (T18430) to (107.33, 121.16, 19.3) mm, rotated rx 180 ry 0 rz -180 deg; joints [1.888, 67.7, -31.262, 3.176, -36.479, -2.555]
  Call Extruder 0.04317
  MoveL (T18431) to (108.32, 120.16, 19.3) mm, rotated rx 180 ry 0 rz -180 deg; joints [1.888, 67.7, -31.262, 3.176, -36.479, -2.555]
  Call Extruder 0.01786
  MoveL (T18432) to (107.74, 120.16, 19.3) mm, rotated rx 180 ry 0 rz -180 deg; joints [1.884, 67.958, -31.748, 3.187, -36.253, -2.571]
  Call Extruder 0.04317
  MoveL (T18433) to (106.75, 121.16, 19.3) mm, rotated rx 180 ry 0 rz -180 deg; joints [1.875, 68.013, -31.85, 3.175, -36.204, -2.563]
  Call Extruder 0.01786
  MoveL (T18434) to (106.17, 121.16, 19.3) mm, rotated rx 180 ry 0 rz -180 deg; joints [1.875, 68.013, -31.85, 3.175, -36.204, -2.563]
  Call Extruder 0.06059
  MoveL (T18435) to (107.56, 119.76, 19.3) mm, rotated rx 180 ry 0 rz -180 deg; joints [1.875, 68.013, -31.85, 3.175, -36.204, -2.563]
  Call Extruder 0.01786
  MoveL (T18436) to (107.56, 119.18, 19.3) mm, rotated rx 180 ry 0 rz -180 deg; joints [1.775, 68.255, -32.305, 3.021, -35.988, -2.445]
  Call Extruder 0.08584
  MoveL (T18437) to (105.59, 121.16, 19.3) mm, rotated rx 180 ry 0 rz -180 deg; joints [1.775, 68.255, -32.305, 3.021, -35.988, -2.445]
  Call Extruder 0.01786
  MoveL (T18438) to (105.01, 121.16, 19.3) mm, rotated rx 180 ry 0 rz -180 deg; joints [1.775, 68.255, -32.305, 3.021, -35.988, -2.445]
  Call Extruder 0.1111
  MoveL (T18439) to (107.56, 118.6, 19.3) mm, rotated rx 180 ry 0 rz -180 deg; joints [2.29, 69.746, -35.106, 4.024, -34.706, -3.31]
  Call Extruder 0.01786
  MoveL (T18440) to (107.56, 118.02, 19.3) mm, rotated rx 180 ry 0 rz -180 deg; joints [2.29, 69.746, -35.106, 4.024, -34.706, -3.31]
  Call Extruder 0.13635
  MoveL (T18441) to (104.42, 121.16, 19.3) mm, rotated rx 180 ry 0 rz -180 deg; joints [2.29, 69.746, -35.106, 4.024, -34.706, -3.31]
  Call Extruder 0.01786
  MoveL (T18442) to (103.84, 121.16, 19.3) mm, rotated rx 180 ry 0 rz -180 deg; joints [2.356, 69.753, -35.12, 4.14, -34.703, -3.405]
  Call Extruder 0.1616
  MoveL (T18443) to (107.56, 117.44, 19.3) mm, rotated rx 180 ry 0 rz -180 deg; joints [2.356, 69.753, -35.12, 4.14, -34.703, -3.405]
  Call Extruder 0.01786
  MoveL (T18444) to (107.56, 116.86, 19.3) mm, rotated rx 180 ry 0 rz -180 deg; joints [2.356, 69.753, -35.12, 4.14, -34.703, -3.405]
  Call Extruder 0.1616
  MoveL (T18445) to (103.84, 120.58, 19.3) mm, rotated rx 180 ry 0 rz -180 deg; joints [2.356, 69.753, -35.12, 4.14, -34.703, -3.405]
  Call Extruder 0.01786
  MoveL (T18446) to (103.84, 119.99, 19.3) mm, rotated rx 180 ry 0 rz -180 deg; joints [3.288, 67.515, -30.916, 5.503, -36.726, -4.416]
  Call Extruder 0.29173
  MoveL (T18447) to (110.56, 113.28, 19.3) mm, rotated rx 180 ry 0 rz -180 deg; joints [3.288, 67.515, -30.916, 5.503, -36.726, -4.416]
  Call Extruder 0.01328
  MoveL (T18448) to (110.36, 112.9, 19.3) mm, rotated rx 180 ry 0 rz -180 deg; joints [3.288, 67.515, -30.916, 5.503, -36.726, -4.416]
  Call Extruder 0.2832
  MoveL (T18449) to (103.84, 119.41, 19.3) mm, rotated rx 180 ry 0 rz -180 deg; joints [3.295, 67.217, -30.356, 5.481, -36.987, -4.383]
  Call Extruder 0.01786
  MoveL (T18450) to (103.84, 118.83, 19.3) mm, rotated rx 180 ry 0 rz -180 deg; joints [3.295, 67.217, -30.356, 5.481, -36.987, -4.383]
  Call Extruder 0.27467
  MoveL (T18451) to (110.16, 112.51, 19.3) mm, rotated rx 180 ry 0 rz -180 deg; joints [3.295, 67.217, -30.356, 5.481, -36.987, -4.383]
  Call Extruder 0.01328
  MoveL (T18452) to (109.97, 112.13, 19.3) mm, rotated rx 180 ry 0 rz -180 deg; joints [3.295, 67.217, -30.356, 5.481, -36.987, -4.383]
  Call Extruder 0.26614
  MoveL (T18453) to (103.84, 118.25, 19.3) mm, rotated rx 180 ry 0 rz -180 deg; joints [2.938, 66.251, -28.543, 4.797, -37.806, -3.793]
  Call Extruder 0.01786
  MoveL (T18454) to (103.84, 117.67, 19.3) mm, rotated rx 180 ry 0 rz -180 deg; joints [2.938, 66.251, -28.543, 4.797, -37.806, -3.793]
  Call Extruder 0.25761
  MoveL (T18455) to (109.77, 111.74, 19.3) mm, rotated rx 180 ry 0 rz -180 deg; joints [2.938, 66.251, -28.543, 4.797, -37.806, -3.793]
  Call Extruder 0.01328
  MoveL (T18456) to (109.57, 111.36, 19.3) mm, rotated rx 180 ry 0 rz -180 deg; joints [2.818, 66.237, -28.516, 4.6, -37.81, -3.637]
  Call Extruder 0.24908
  MoveL (T18457) to (103.84, 117.09, 19.3) mm, rotated rx 180 ry 0 rz -180 deg; joints [2.818, 66.237, -28.516, 4.6, -37.81, -3.637]
  Call Extruder 0.01786
  MoveL (T18458) to (103.84, 116.51, 19.3) mm, rotated rx 180 ry 0 rz -180 deg; joints [1.815, 68.554, -32.866, 3.109, -35.727, -2.525]
  Call Extruder 0.24055
  MoveL (T18459) to (109.38, 110.97, 19.3) mm, rotated rx 180 ry 0 rz -180 deg; joints [1.815, 68.554, -32.866, 3.109, -35.727, -2.525]
  Call Extruder 0.01328
  MoveL (T18460) to (109.18, 110.59, 19.3) mm, rotated rx 180 ry 0 rz -180 deg; joints [1.866, 68.698, -33.138, 3.206, -35.603, -2.608]
  Call Extruder 0.23202
  MoveL (T18461) to (103.84, 115.93, 19.3) mm, rotated rx 180 ry 0 rz -180 deg; joints [1.866, 68.698, -33.138, 3.206, -35.603, -2.608]
  Call Extruder 0.01786
  MoveL (T18462) to (103.84, 115.35, 19.3) mm, rotated rx 180 ry 0 rz -180 deg; joints [1.874, 68.756, -33.247, 3.224, -35.552, -2.624]
  Call Extruder 0.22349
  MoveL (T18463) to (108.98, 110.21, 19.3) mm, rotated rx 180 ry 0 rz -180 deg; joints [1.874, 68.756, -33.247, 3.224, -35.552, -2.624]
  Call Extruder 0.01328
  MoveL (T18464) to (108.79, 109.82, 19.3) mm, rotated rx 180 ry 0 rz -180 deg; joints [1.874, 68.756, -33.247, 3.224, -35.552, -2.624]
  Call Extruder 0.21496
  MoveL (T18465) to (103.84, 114.77, 19.3) mm, rotated rx 180 ry 0 rz -180 deg; joints [1.869, 69.192, -34.065, 3.246, -35.17, -2.654]
  Call Extruder 0.01786
  MoveL (T18466) to (103.84, 114.18, 19.3) mm, rotated rx 180 ry 0 rz -180 deg; joints [1.869, 69.192, -34.065, 3.246, -35.17, -2.654]
  Call Extruder 0.20642
  MoveL (T18467) to (108.59, 109.44, 19.3) mm, rotated rx 180 ry 0 rz -180 deg; joints [1.869, 69.192, -34.065, 3.246, -35.17, -2.654]
  Call Extruder 0.01328
  MoveL (T18468) to (108.4, 109.05, 19.3) mm, rotated rx 180 ry 0 rz -180 deg; joints [1.869, 69.192, -34.065, 3.246, -35.17, -2.654]
  Call Extruder 0.19789
  MoveL (T18469) to (103.84, 113.6, 19.3) mm, rotated rx 180 ry 0 rz -180 deg; joints [1.869, 69.192, -34.065, 3.246, -35.17, -2.654]
  Call Extruder 0.01786
  MoveL (T18470) to (103.84, 113.02, 19.3) mm, rotated rx 180 ry 0 rz -180 deg; joints [1.869, 69.192, -34.065, 3.246, -35.17, -2.654]
  Call Extruder 0.18936
  MoveL (T18471) to (108.2, 108.67, 19.3) mm, rotated rx 180 ry 0 rz -180 deg; joints [1.869, 69.192, -34.065, 3.246, -35.17, -2.654]
  Call Extruder 0.01328
  MoveL (T18472) to (108, 108.28, 19.3) mm, rotated rx 180 ry 0 rz -180 deg; joints [1.869, 69.192, -34.065, 3.246, -35.17, -2.654]
  Call Extruder 0.18083
  MoveL (T18473) to (103.84, 112.44, 19.3) mm, rotated rx 180 ry 0 rz -180 deg; joints [1.869, 69.192, -34.065, 3.246, -35.17, -2.654]
  Call Extruder 0.01786
  MoveL (T18474) to (103.84, 111.86, 19.3) mm, rotated rx 180 ry 0 rz -180 deg; joints [1.869, 69.192, -34.065, 3.246, -35.17, -2.654]
  Call Extruder 0.1723
  MoveL (T18475) to (107.81, 107.9, 19.3) mm, rotated rx 180 ry 0 rz -180 deg; joints [1.873, 68.885, -33.49, 3.231, -35.439, -2.633]
  Call Extruder 0.01328
  MoveL (T18476) to (107.61, 107.51, 19.3) mm, rotated rx 180 ry 0 rz -180 deg; joints [1.873, 68.885, -33.49, 3.231, -35.439, -2.633]
  Call Extruder 0.16377
  MoveL (T18477) to (103.84, 111.28, 19.3) mm, rotated rx 180 ry 0 rz -180 deg; joints [1.873, 68.885, -33.49, 3.231, -35.439, -2.633]
  Call Extruder 0.01786
  MoveL (T18478) to (103.84, 110.7, 19.3) mm, rotated rx 180 ry 0 rz -180 deg; joints [1.873, 68.885, -33.49, 3.231, -35.439, -2.633]
  Call Extruder 0.15795
  MoveL (T18479) to (107.48, 107.07, 19.3) mm, rotated rx 180 ry 0 rz -180 deg; joints [1.873, 68.885, -33.49, 3.231, -35.439, -2.633]
  Call Extruder 0.01786
  MoveL (T18480) to (107.48, 106.48, 19.3) mm, rotated rx 180 ry 0 rz -180 deg; joints [1.873, 68.885, -33.49, 3.231, -35.439, -2.633]
  Call Extruder 0.15795
  MoveL (T18481) to (103.84, 110.12, 19.3) mm, rotated rx 180 ry 0 rz -180 deg; joints [1.873, 68.885, -33.49, 3.231, -35.439, -2.633]
  Call Extruder 0.01786
  MoveL (T18482) to (103.84, 109.54, 19.3) mm, rotated rx 180 ry 0 rz -180 deg; joints [1.873, 68.885, -33.49, 3.231, -35.439, -2.633]
  Call Extruder 0.16591
  MoveL (T18483) to (107.66, 105.72, 19.3) mm, rotated rx 180 ry 0 rz -180 deg; joints [1.873, 68.652, -33.451, 3.246, -35.245, -2.652]
  Set speed (45.0 mm/s)
  Call Extruder -1.6
  MoveL (T18484) to (107.66, 105.72, 19.3) mm, rotated rx 180 ry 0 rz -180 deg; joints [1.652, 70.777, -37.438, 3.005, -33.375, -2.51]
  Set speed (120.0 mm/s)
  MoveL (T18485) to (107.66, 105.72, 19.3) mm, rotated rx 180 ry 0 rz -180 deg; joints [1.652, 71.009, -37.48, 2.99, -33.565, -2.492]
  Call Extruder -0.38
  MoveL (T18486) to (106.91, 106.47, 19.3) mm, rotated rx 180 ry 0 rz -180 deg; joints [1.652, 71.009, -37.48, 2.99, -33.565, -2.492]
  Set speed (45.0 mm/s)
  Call Extruder -0.02
  MoveL (T18487) to (106.91, 106.47, 19.3) mm, rotated rx 180 ry 0 rz -180 deg; joints [1.652, 71.009, -37.48, 2.99, -33.565, -2.492]
  Set speed (150.0 mm/s)
  MoveL (T18488) to (106.91, 106.47, 21.3) mm, rotated rx 180 ry 0 rz -180 deg; joints [1.652, 71.009, -37.48, 2.99, -33.565, -2.492]
  MoveL (T18489) to (109.14, 103.66, 21.3) mm, rotated rx 180 ry 0 rz -180 deg; joints [1.652, 71.009, -37.48, 2.99, -33.565, -2.492]
  MoveL (T18490) to (109.14, 103.66, 19.3) mm, rotated rx 180 ry 0 rz -180 deg; joints [1.652, 71.009, -37.48, 2.99, -33.565, -2.492]
  Set speed (40.0 mm/s)
  Call Extruder 2.0
  MoveL (T18491) to (109.14, 103.66, 19.3) mm, rotated rx 180 ry 0 rz -180 deg; joints [1.396, 70.989, -37.442, 2.525, -33.573, -2.104]
  Call Extruder 0.23019
  MoveL (T18492) to (103.84, 108.96, 19.3) mm, rotated rx 180 ry 0 rz -180 deg; joints [1.396, 70.989, -37.442, 2.525, -33.573, -2.104]
  Call Extruder 0.01786
  MoveL (T18493) to (103.84, 108.38, 19.3) mm, rotated rx 180 ry 0 rz -180 deg; joints [1.396, 70.989, -37.442, 2.525, -33.573, -2.104]
  Call Extruder 0.19697
  MoveL (T18494) to (108.38, 103.84, 19.3) mm, rotated rx 180 ry 0 rz -180 deg; joints [1.396, 70.989, -37.442, 2.525, -33.573, -2.104]
  Call Extruder 0.01786
  MoveL (T18495) to (107.79, 103.84, 19.3) mm, rotated rx 180 ry 0 rz -180 deg; joints [1.467, 70.79, -37.068, 2.64, -33.75, -2.196]
  Call Extruder 0.17171
  MoveL (T18496) to (103.84, 107.79, 19.3) mm, rotated rx 180 ry 0 rz -180 deg; joints [1.467, 70.79, -37.068, 2.64, -33.75, -2.196]
  Call Extruder 0.01786
  MoveL (T18497) to (103.84, 107.21, 19.3) mm, rotated rx 180 ry 0 rz -180 deg; joints [1.467, 70.79, -37.068, 2.64, -33.75, -2.196]
  Call Extruder 0.14646
  MoveL (T18498) to (107.21, 103.84, 19.3) mm, rotated rx 180 ry 0 rz -180 deg; joints [1.607, 70.801, -37.088, 2.893, -33.746, -2.406]
  Call Extruder 0.01786
  MoveL (T18499) to (106.63, 103.84, 19.3) mm, rotated rx 180 ry 0 rz -180 deg; joints [1.607, 70.801, -37.088, 2.893, -33.746, -2.406]
  Call Extruder 0.1212
  MoveL (T18500) to (103.84, 106.63, 19.3) mm, rotated rx 180 ry 0 rz -180 deg; joints [1.607, 70.801, -37.088, 2.893, -33.746, -2.406]
  Call Extruder 0.01786
  MoveL (T18501) to (103.84, 106.05, 19.3) mm, rotated rx 180 ry 0 rz -180 deg; joints [1.628, 70.777, -37.043, 2.93, -33.768, -2.436]
  Call Extruder 0.09595
  MoveL (T18502) to (106.05, 103.84, 19.3) mm, rotated rx 180 ry 0 rz -180 deg; joints [1.628, 70.777, -37.043, 2.93, -33.768, -2.436]
  Call Extruder 0.01786
  MoveL (T18503) to (105.47, 103.84, 19.3) mm, rotated rx 180 ry 0 rz -180 deg; joints [1.628, 70.777, -37.043, 2.93, -33.768, -2.436]
  Call Extruder 0.07069
  MoveL (T18504) to (103.84, 105.47, 19.3) mm, rotated rx 180 ry 0 rz -180 deg; joints [1.628, 70.777, -37.043, 2.93, -33.768, -2.436]
  Call Extruder 0.01786
  MoveL (T18505) to (103.84, 104.89, 19.3) mm, rotated rx 180 ry 0 rz -180 deg; joints [1.628, 70.777, -37.043, 2.93, -33.768, -2.436]
  Call Extruder 0.04544
  MoveL (T18506) to (104.89, 103.84, 19.3) mm, rotated rx 180 ry 0 rz -180 deg; joints [1.659, 70.692, -36.884, 2.979, -33.844, -2.475]
  Call Extruder 0.01786
  MoveL (T18507) to (104.31, 103.84, 19.3) mm, rotated rx 180 ry 0 rz -180 deg; joints [1.763, 71.019, -37.498, 3.19, -33.562, -2.659]
  Call Extruder 0.02815
  MoveL (T18508) to (103.66, 104.49, 19.3) mm, rotated rx 180 ry 0 rz -180 deg; joints [1.763, 71.019, -37.498, 3.19, -33.562, -2.659]
  Set speed (45.0 mm/s)
  Call Extruder -1.6
  MoveL (T18509) to (103.66, 104.49, 19.3) mm, rotated rx 180 ry 0 rz -180 deg; joints [1.787, 71.021, -37.503, 3.234, -33.561, -2.695]
  Set speed (120.0 mm/s)
  MoveL (T18510) to (103.66, 104.49, 19.3) mm, rotated rx 180 ry 0 rz -180 deg; joints [1.787, 71.021, -37.503, 3.234, -33.561, -2.695]
  Call Extruder -0.3262
  MoveL (T18511) to (104.31, 103.84, 19.3) mm, rotated rx 180 ry 0 rz -180 deg; joints [1.787, 71.021, -37.503, 3.234, -33.561, -2.695]
  Call Extruder -0.0538
  MoveL (T18512) to (104.46, 103.84, 19.3) mm, rotated rx 180 ry 0 rz -180 deg; joints [1.794, 70.393, -36.321, 3.199, -34.113, -2.65]
  Set speed (45.0 mm/s)
  Call Extruder -0.02
  MoveL (T18513) to (104.46, 103.84, 19.3) mm, rotated rx 180 ry 0 rz -180 deg; joints [1.794, 70.393, -36.321, 3.199, -34.113, -2.65]
  Set speed (150.0 mm/s)
  MoveL (T18514) to (104.46, 103.84, 21.3) mm, rotated rx 180 ry 0 rz -180 deg; joints [1.803, 70.332, -36.208, 3.211, -34.166, -2.658]
  MoveL (T18515) to (109.4, 105.47, 21.3) mm, rotated rx 180 ry 0 rz -180 deg; joints [1.803, 70.332, -36.208, 3.211, -34.166, -2.658]
  MoveL (T18516) to (109.4, 105.47, 19.5) mm, rotated rx 180 ry 0 rz -180 deg; joints [1.803, 70.332, -36.208, 3.211, -34.166, -2.658]
  Set speed (40.0 mm/s)
  Call Extruder 2.0
  MoveL (T18517) to (109.4, 105.47, 19.5) mm, rotated rx 180 ry 0 rz -180 deg; joints [1.803, 70.332, -36.208, 3.211, -34.166, -2.658]
  Call Extruder 0.25145
  MoveL (T18518) to (117.65, 105.47, 19.5) mm, rotated rx 180 ry 0 rz -180 deg; joints [1.915, 70.033, -35.646, 3.387, -34.434, -2.795]
  Call Extruder 0.10939
  MoveL (T18519) to (117.65, 109.06, 19.5) mm, rotated rx 180 ry 0 rz -180 deg; joints [1.861, 69.871, -35.341, 3.281, -34.574, -2.702]
  Call Extruder 0.14732
  MoveL (T18520) to (112.81, 109.06, 19.5) mm, rotated rx 180 ry 0 rz -180 deg; joints [1.861, 69.871, -35.341, 3.281, -34.574, -2.702]
  Call Extruder 0.31102
  MoveL (T18521) to (117.47, 118.15, 19.5) mm, rotated rx 180 ry 0 rz -180 deg; joints [1.861, 69.871, -35.341, 3.281, -34.574, -2.702]
  Call Extruder 0.05209
  MoveL (T18522) to (117.47, 119.86, 19.5) mm, rotated rx 180 ry 0 rz -180 deg; joints [1.863, 69.719, -35.055, 3.273, -34.707, -2.691]
  Call Extruder 0.29244
  MoveL (T18523) to (107.87, 119.86, 19.5) mm, rotated rx 180 ry 0 rz -180 deg; joints [1.863, 69.719, -35.055, 3.273, -34.707, -2.691]
  Call Extruder 0.10939
  MoveL (T18524) to (107.87, 116.27, 19.5) mm, rotated rx 180 ry 0 rz -180 deg; joints [3.316, 66.3, -28.635, 5.417, -37.789, -4.286]
  Call Extruder 0.13869
  MoveL (T18525) to (112.42, 116.27, 19.5) mm, rotated rx 180 ry 0 rz -180 deg; joints [3.316, 66.3, -28.635, 5.417, -37.789, -4.286]
  Call Extruder 0.31084
  MoveL (T18526) to (107.78, 107.18, 19.5) mm, rotated rx 180 ry 0 rz -180 deg; joints [3.316, 66.3, -28.635, 5.417, -37.789, -4.286]
  Call Extruder 0.05206
  MoveL (T18527) to (107.78, 105.47, 19.5) mm, rotated rx 180 ry 0 rz -180 deg; joints [3.301, 66.938, -29.832, 5.461, -37.231, -4.353]
  Call Extruder 0.04735
  MoveL (T18528) to (109.34, 105.47, 19.5) mm, rotated rx 180 ry 0 rz -180 deg; joints [3.301, 66.938, -29.832, 5.461, -37.231, -4.353]
  Set speed (150.0 mm/s)
  MoveL (T18529) to (109, 105.88, 19.5) mm, rotated rx 180 ry 0 rz -180 deg; joints [3.301, 66.938, -29.832, 5.461, -37.231, -4.353]
  Set speed (40.0 mm/s)
  MoveL (T18530) to (109, 105.88, 19.5) mm, rotated rx 180 ry 0 rz -180 deg; joints [3.301, 66.938, -29.832, 5.461, -37.231, -4.353]
  Call Extruder 0.25124
  MoveL (T18531) to (117.24, 105.88, 19.5) mm, rotated rx 180 ry 0 rz -180 deg; joints [3.301, 66.938, -29.832, 5.461, -37.231, -4.353]
  Call Extruder 0.08459
  MoveL (T18532) to (117.24, 108.65, 19.5) mm, rotated rx 180 ry 0 rz -180 deg; joints [3.301, 66.938, -29.832, 5.461, -37.231, -4.353]
  Call Extruder 0.1552
  MoveL (T18533) to (112.15, 108.65, 19.5) mm, rotated rx 180 ry 0 rz -180 deg; joints [3.301, 66.938, -29.832, 5.461, -37.231, -4.353]
  Call Extruder 0.32831
  MoveL (T18534) to (117.06, 118.25, 19.5) mm, rotated rx 180 ry 0 rz -180 deg; joints [3.301, 66.938, -29.832, 5.461, -37.231, -4.353]
  Call Extruder 0.0367
  MoveL (T18535) to (117.06, 119.45, 19.5) mm, rotated rx 180 ry 0 rz -180 deg; joints [3.301, 66.938, -29.832, 5.461, -37.231, -4.353]
  Call Extruder 0.26763
  MoveL (T18536) to (108.27, 119.45, 19.5) mm, rotated rx 180 ry 0 rz -180 deg; joints [3.301, 66.938, -29.832, 5.461, -37.231, -4.353]
  Call Extruder 0.08459
  MoveL (T18537) to (108.27, 116.67, 19.5) mm, rotated rx 180 ry 0 rz -180 deg; joints [3.301, 66.938, -29.832, 5.461, -37.231, -4.353]
  Call Extruder 0.14654
  MoveL (T18538) to (113.08, 116.67, 19.5) mm, rotated rx 180 ry 0 rz -180 deg; joints [3.308, 66.658, -29.306, 5.441, -37.477, -4.323]
  Call Extruder 0.32811
  MoveL (T18539) to (108.19, 107.08, 19.5) mm, rotated rx 180 ry 0 rz -180 deg; joints [3.308, 66.658, -29.306, 5.441, -37.477, -4.323]
  Call Extruder 0.03668
  MoveL (T18540) to (108.19, 105.88, 19.5) mm, rotated rx 180 ry 0 rz -180 deg; joints [3.308, 66.658, -29.306, 5.441, -37.477, -4.323]
  Call Extruder 0.02276
  MoveL (T18541) to (108.94, 105.88, 19.5) mm, rotated rx 180 ry 0 rz -180 deg; joints [3.308, 66.658, -29.306, 5.441, -37.477, -4.323]
  Set speed (150.0 mm/s)
  MoveL (T18542) to (108.6, 106.28, 19.5) mm, rotated rx 180 ry 0 rz -180 deg; joints [3.308, 66.658, -29.306, 5.441, -37.477, -4.323]
  Set speed (25.0 mm/s)
  MoveL (T18543) to (108.6, 106.28, 19.5) mm, rotated rx 180 ry 0 rz -180 deg; joints [3.308, 66.658, -29.306, 5.441, -37.477, -4.323]
  Call Extruder 0.25102
  MoveL (T18544) to (116.84, 106.28, 19.5) mm, rotated rx 180 ry 0 rz -180 deg; joints [3.308, 66.658, -29.306, 5.441, -37.477, -4.323]
  Call Extruder 0.05979
  MoveL (T18545) to (116.84, 108.25, 19.5) mm, rotated rx 180 ry 0 rz -180 deg; joints [3.308, 66.422, -29.27, 5.466, -37.278, -4.354]
  Call Extruder 0.16307
  MoveL (T18546) to (111.48, 108.25, 19.5) mm, rotated rx 180 ry 0 rz -180 deg; joints [3.308, 66.422, -29.27, 5.466, -37.278, -4.354]
  Call Extruder 0.3456
  MoveL (T18547) to (116.65, 118.34, 19.5) mm, rotated rx 180 ry 0 rz -180 deg; joints [1.407, 66.005, -28.487, 2.31, -37.54, -1.832]
  Call Extruder 0.02131
  MoveL (T18548) to (116.65, 119.04, 19.5) mm, rotated rx 180 ry 0 rz -180 deg; joints [1.407, 66.005, -28.487, 2.31, -37.54, -1.832]
  Call Extruder 0.24283
  MoveL (T18549) to (108.68, 119.04, 19.5) mm, rotated rx 180 ry 0 rz -180 deg; joints [1.407, 66.217, -28.52, 2.301, -37.72, -1.82]
  Call Extruder 0.05979
  MoveL (T18550) to (108.68, 117.08, 19.5) mm, rotated rx 180 ry 0 rz -180 deg; joints [1.407, 66.217, -28.52, 2.301, -37.72, -1.82]
  Call Extruder 0.15438
  MoveL (T18551) to (113.75, 117.08, 19.5) mm, rotated rx 180 ry 0 rz -180 deg; joints [1.407, 66.217, -28.52, 2.301, -37.72, -1.82]
  Call Extruder 0.34538
  MoveL (T18552) to (108.6, 106.98, 19.5) mm, rotated rx 180 ry 0 rz -180 deg; joints [1.407, 66.217, -28.52, 2.301, -37.72, -1.82]
  Call Extruder 0.01947
  MoveL (T18553) to (108.6, 106.34, 19.5) mm, rotated rx 180 ry 0 rz -180 deg; joints [1.407, 66.217, -28.52, 2.301, -37.72, -1.82]
  Set speed (150.0 mm/s)
  MoveL (T18554) to (108.54, 105.89, 19.5) mm, rotated rx 180 ry 0 rz -180 deg; joints [1.407, 66.217, -28.52, 2.301, -37.72, -1.82]
  Set speed (45.0 mm/s)
  Call Extruder -1.6
  MoveL (T18555) to (108.54, 105.89, 19.5) mm, rotated rx 180 ry 0 rz -180 deg; joints [1.407, 66.217, -28.52, 2.301, -37.72, -1.82]
  Set speed (120.0 mm/s)
  MoveL (T18556) to (108.54, 105.89, 19.5) mm, rotated rx 180 ry 0 rz -180 deg; joints [1.363, 71.059, -37.612, 2.472, -33.471, -2.063]
  Call Extruder -0.38
  MoveL (T18557) to (109.66, 106.33, 19.5) mm, rotated rx 180 ry 0 rz -180 deg; joints [1.363, 71.059, -37.612, 2.472, -33.471, -2.063]
  Set speed (45.0 mm/s)
  Call Extruder -0.02
  MoveL (T18558) to (109.66, 106.33, 19.5) mm, rotated rx 180 ry 0 rz -180 deg; joints [3.241, 71.286, -38.039, 5.898, -33.386, -4.93]
  Set speed (150.0 mm/s)
  MoveL (T18559) to (109.66, 106.33, 21.5) mm, rotated rx 180 ry 0 rz -180 deg; joints [3.241, 71.286, -38.039, 5.898, -33.386, -4.93]
  MoveL (T18560) to (104.34, 103.54, 21.5) mm, rotated rx 180 ry 0 rz -180 deg; joints [3.241, 71.286, -38.039, 5.898, -33.386, -4.93]
  MoveL (T18561) to (104.34, 103.54, 19.5) mm, rotated rx 180 ry 0 rz -180 deg; joints [3.351, 66.203, -28.493, 5.468, -37.837, -4.324]
  Set speed (40.0 mm/s)
  Call Extruder 2.0
  MoveL (T18562) to (104.34, 103.54, 19.5) mm, rotated rx 180 ry 0 rz -180 deg; joints [3.351, 66.203, -28.493, 5.468, -37.837, -4.324]
  Call Extruder 0.52159
  MoveL (T18563) to (121.46, 103.54, 19.5) mm, rotated rx 180 ry 0 rz -180 deg; joints [3.351, 66.203, -28.493, 5.468, -37.837, -4.324]
  Call Extruder 0.54596
  MoveL (T18564) to (121.46, 121.46, 19.5) mm, rotated rx 180 ry 0 rz -180 deg; joints [3.351, 66.203, -28.493, 5.468, -37.837, -4.324]
  Call Extruder 0.54596
  MoveL (T18565) to (103.54, 121.46, 19.5) mm, rotated rx 180 ry 0 rz -180 deg; joints [1.409, 66.012, -28.134, 2.295, -37.9, -1.811]
  Call Extruder 0.54596
  MoveL (T18566) to (103.54, 103.54, 19.5) mm, rotated rx 180 ry 0 rz -180 deg; joints [1.409, 66.012, -28.134, 2.295, -37.9, -1.811]
  Call Extruder 0.02254
  MoveL (T18567) to (104.28, 103.54, 19.5) mm, rotated rx 180 ry 0 rz -180 deg; joints [1.409, 66.012, -28.134, 2.295, -37.9, -1.811]
  Set speed (150.0 mm/s)
  MoveL (T18568) to (103.53, 103.13, 19.5) mm, rotated rx 180 ry 0 rz -180 deg; joints [1.409, 66.012, -28.134, 2.295, -37.9, -1.811]
  Set speed (40.0 mm/s)
  MoveL (T18569) to (103.53, 103.13, 19.5) mm, rotated rx 180 ry 0 rz -180 deg; joints [1.409, 66.012, -28.134, 2.295, -37.9, -1.811]
  Call Extruder 0.55858
  MoveL (T18570) to (121.87, 103.13, 19.5) mm, rotated rx 180 ry 0 rz -180 deg; joints [1.407, 66.202, -28.491, 2.3, -37.733, -1.82]
  Call Extruder 0.57077
  MoveL (T18571) to (121.87, 121.87, 19.5) mm, rotated rx 180 ry 0 rz -180 deg; joints [1.365, 66.007, -28.126, 2.223, -37.902, -1.754]
  Call Extruder 0.57077
  MoveL (T18572) to (103.13, 121.87, 19.5) mm, rotated rx 180 ry 0 rz -180 deg; joints [1.365, 66.007, -28.126, 2.223, -37.902, -1.754]
  Call Extruder 0.57077
  MoveL (T18573) to (103.13, 103.13, 19.5) mm, rotated rx 180 ry 0 rz -180 deg; joints [1.365, 66.007, -28.126, 2.223, -37.902, -1.754]
  Call Extruder 0.01036
  MoveL (T18574) to (103.47, 103.13, 19.5) mm, rotated rx 180 ry 0 rz -180 deg; joints [1.365, 66.007, -28.126, 2.223, -37.902, -1.754]
  Set speed (150.0 mm/s)
  MoveL (T18575) to (102.72, 102.81, 19.5) mm, rotated rx 180 ry 0 rz -180 deg; joints [1.319, 71.184, -37.847, 2.4, -33.36, -2.005]
  Set speed (25.0 mm/s)
  MoveL (T18576) to (102.72, 102.81, 19.5) mm, rotated rx 180 ry 0 rz -180 deg; joints [1.319, 71.184, -37.847, 2.4, -33.36, -2.005]
  Call Extruder 0.00259
  MoveL (T18577) to (102.72, 102.72, 19.5) mm, rotated rx 180 ry 0 rz -180 deg; joints [1.319, 71.184, -37.847, 2.4, -33.36, -2.005]
  Call Extruder 0.59557
  MoveL (T18578) to (122.28, 102.72, 19.5) mm, rotated rx 180 ry 0 rz -180 deg; joints [3.282, 71.423, -38.296, 5.989, -33.27, -5.013]
  Call Extruder 0.59557
  MoveL (T18579) to (122.28, 122.28, 19.5) mm, rotated rx 180 ry 0 rz -180 deg; joints [3.282, 71.423, -38.296, 5.989, -33.27, -5.013]
  Call Extruder 0.59557
  MoveL (T18580) to (102.72, 122.28, 19.5) mm, rotated rx 180 ry 0 rz -180 deg; joints [3.282, 71.423, -38.296, 5.989, -33.27, -5.013]
  Call Extruder 0.59115
  MoveL (T18581) to (102.72, 102.87, 19.5) mm, rotated rx 180 ry 0 rz -180 deg; joints [3.398, 66.104, -28.308, 5.533, -37.926, -4.37]
  Set speed (150.0 mm/s)
  MoveL (T18582) to (102.78, 102.75, 19.5) mm, rotated rx 180 ry 0 rz -180 deg; joints [3.398, 66.104, -28.308, 5.533, -37.926, -4.37]
  Set speed (45.0 mm/s)
  Call Extruder -1.6
  MoveL (T18583) to (102.78, 102.75, 19.5) mm, rotated rx 180 ry 0 rz -180 deg; joints [3.398, 66.104, -28.308, 5.533, -37.926, -4.37]
  Set speed (120.0 mm/s)
  MoveL (T18584) to (102.78, 102.75, 19.5) mm, rotated rx 180 ry 0 rz -180 deg; joints [1.366, 65.905, -27.934, 2.22, -37.992, -1.75]
  Call Extruder -0.05166
  MoveL (T18585) to (102.72, 102.72, 19.5) mm, rotated rx 180 ry 0 rz -180 deg; joints [1.366, 65.905, -27.934, 2.22, -37.992, -1.75]
  Call Extruder -0.32834
  MoveL (T18586) to (103.65, 102.72, 19.5) mm, rotated rx 180 ry 0 rz -180 deg; joints [1.366, 65.905, -27.934, 2.22, -37.992, -1.75]
  Set speed (45.0 mm/s)
  Call Extruder -0.02
  MoveL (T18587) to (103.65, 102.72, 19.5) mm, rotated rx 180 ry 0 rz -180 deg; joints [1.366, 65.905, -27.934, 2.22, -37.992, -1.75]
  Set speed (150.0 mm/s)
  MoveL (T18588) to (103.65, 102.72, 21.5) mm, rotated rx 180 ry 0 rz -180 deg; joints [1.365, 65.992, -28.097, 2.222, -37.916, -1.754]
  MoveL (T18589) to (120.51, 103.66, 21.5) mm, rotated rx 180 ry 0 rz -180 deg; joints [1.365, 65.992, -28.097, 2.222, -37.916, -1.754]
  MoveL (T18590) to (120.51, 103.66, 19.5) mm, rotated rx 180 ry 0 rz -180 deg; joints [1.365, 65.992, -28.097, 2.222, -37.916, -1.754]
  Set speed (40.0 mm/s)
  Call Extruder 2.0
  MoveL (T18591) to (120.51, 103.66, 19.5) mm, rotated rx 180 ry 0 rz -180 deg; joints [1.365, 65.992, -28.097, 2.222, -37.916, -1.754]
  Call Extruder 0.02815
  MoveL (T18592) to (121.16, 104.31, 19.5) mm, rotated rx 180 ry 0 rz -180 deg; joints [1.365, 65.992, -28.097, 2.222, -37.916, -1.754]
  Call Extruder 0.01786
  MoveL (T18593) to (121.16, 104.89, 19.5) mm, rotated rx 180 ry 0 rz -180 deg; joints [1.332, 65.8, -27.736, 2.161, -38.083, -1.701]
  Call Extruder 0.04544
  MoveL (T18594) to (120.11, 103.84, 19.5) mm, rotated rx 180 ry 0 rz -180 deg; joints [1.332, 65.8, -27.736, 2.161, -38.083, -1.701]
  Call Extruder 0.01786
  MoveL (T18595) to (119.53, 103.84, 19.5) mm, rotated rx 180 ry 0 rz -180 deg; joints [1.332, 65.8, -27.736, 2.161, -38.083, -1.701]
  Call Extruder 0.0707
  MoveL (T18596) to (121.16, 105.47, 19.5) mm, rotated rx 180 ry 0 rz -180 deg; joints [1.332, 65.8, -27.736, 2.161, -38.083, -1.701]
  Call Extruder 0.01786
  MoveL (T18597) to (121.16, 106.05, 19.5) mm, rotated rx 180 ry 0 rz -180 deg; joints [1.332, 65.8, -27.736, 2.161, -38.083, -1.701]
  Call Extruder 0.09595
  MoveL (T18598) to (118.95, 103.84, 19.5) mm, rotated rx 180 ry 0 rz -180 deg; joints [1.323, 65.799, -27.735, 2.146, -38.083, -1.689]
  Call Extruder 0.01786
  MoveL (T18599) to (118.37, 103.84, 19.5) mm, rotated rx 180 ry 0 rz -180 deg; joints [1.276, 71.31, -38.084, 2.328, -33.248, -1.947]
  Call Extruder 0.12121
  MoveL (T18600) to (121.16, 106.63, 19.5) mm, rotated rx 180 ry 0 rz -180 deg; joints [1.276, 71.31, -38.084, 2.328, -33.248, -1.947]
  Call Extruder 0.01786
  MoveL (T18601) to (121.16, 107.21, 19.5) mm, rotated rx 180 ry 0 rz -180 deg; joints [3.322, 71.56, -38.554, 6.082, -33.154, -5.097]
  Call Extruder 0.14646
  MoveL (T18602) to (117.79, 103.84, 19.5) mm, rotated rx 180 ry 0 rz -180 deg; joints [3.322, 71.56, -38.554, 6.082, -33.154, -5.097]
  Call Extruder 0.01786
  MoveL (T18603) to (117.21, 103.84, 19.5) mm, rotated rx 180 ry 0 rz -180 deg; joints [3.445, 66.007, -28.124, 5.598, -38.015, -4.416]
  Call Extruder 0.17172
  MoveL (T18604) to (121.16, 107.79, 19.5) mm, rotated rx 180 ry 0 rz -180 deg; joints [3.445, 66.007, -28.124, 5.598, -38.015, -4.416]
  Call Extruder 0.01786
  MoveL (T18605) to (121.16, 108.38, 19.5) mm, rotated rx 180 ry 0 rz -180 deg; joints [3.445, 66.007, -28.124, 5.598, -38.015, -4.416]
  Call Extruder 0.19697
  MoveL (T18606) to (116.62, 103.84, 19.5) mm, rotated rx 180 ry 0 rz -180 deg; joints [3.445, 66.007, -28.124, 5.598, -38.015, -4.416]
  Call Extruder 0.01786
  MoveL (T18607) to (116.04, 103.84, 19.5) mm, rotated rx 180 ry 0 rz -180 deg; joints [1.339, 65.8, -27.737, 2.171, -38.083, -1.709]
  Call Extruder 0.0573
  MoveL (T18608) to (117.36, 105.16, 19.5) mm, rotated rx 180 ry 0 rz -180 deg; joints [1.339, 65.8, -27.737, 2.171, -38.083, -1.709]
  Call Extruder 0.01786
  MoveL (T18609) to (116.78, 105.16, 19.5) mm, rotated rx 180 ry 0 rz -180 deg; joints [1.339, 65.8, -27.737, 2.171, -38.083, -1.709]
  Call Extruder 0.0573
  MoveL (T18610) to (115.46, 103.84, 19.5) mm, rotated rx 180 ry 0 rz -180 deg; joints [1.339, 65.8, -27.737, 2.171, -38.083, -1.709]
  Call Extruder 0.01786
  MoveL (T18611) to (114.88, 103.84, 19.5) mm, rotated rx 180 ry 0 rz -180 deg; joints [1.339, 65.8, -27.737, 2.171, -38.083, -1.709]
  Call Extruder 0.0573
  MoveL (T18612) to (116.2, 105.16, 19.5) mm, rotated rx 180 ry 0 rz -180 deg; joints [1.326, 65.815, -27.764, 2.15, -38.07, -1.693]
  Call Extruder 0.01786
  MoveL (T18613) to (115.62, 105.16, 19.5) mm, rotated rx 180 ry 0 rz -180 deg; joints [1.326, 65.815, -27.764, 2.15, -38.07, -1.693]
  Call Extruder 0.0573
  MoveL (T18614) to (114.3, 103.84, 19.5) mm, rotated rx 180 ry 0 rz -180 deg; joints [1.326, 65.815, -27.764, 2.15, -38.07, -1.693]
  Call Extruder 0.01786
  MoveL (T18615) to (113.72, 103.84, 19.5) mm, rotated rx 180 ry 0 rz -180 deg; joints [1.326, 65.815, -27.764, 2.15, -38.07, -1.693]
  Call Extruder 0.0573
  MoveL (T18616) to (115.04, 105.16, 19.5) mm, rotated rx 180 ry 0 rz -180 deg; joints [1.326, 65.815, -27.764, 2.15, -38.07, -1.693]
  Call Extruder 0.01786
  MoveL (T18617) to (114.46, 105.16, 19.5) mm, rotated rx 180 ry 0 rz -180 deg; joints [1.326, 65.815, -27.764, 2.15, -38.07, -1.693]
  Call Extruder 0.0573
  MoveL (T18618) to (113.14, 103.84, 19.5) mm, rotated rx 180 ry 0 rz -180 deg; joints [1.326, 65.815, -27.764, 2.15, -38.07, -1.693]
  Call Extruder 0.01786
  MoveL (T18619) to (112.56, 103.84, 19.5) mm, rotated rx 180 ry 0 rz -180 deg; joints [1.326, 65.815, -27.764, 2.15, -38.07, -1.693]
  Call Extruder 0.0573
  MoveL (T18620) to (113.88, 105.16, 19.5) mm, rotated rx 180 ry 0 rz -180 deg; joints [1.326, 65.815, -27.764, 2.15, -38.07, -1.693]
  Call Extruder 0.01786
  MoveL (T18621) to (113.3, 105.16, 19.5) mm, rotated rx 180 ry 0 rz -180 deg; joints [1.326, 65.815, -27.764, 2.15, -38.07, -1.693]
  Call Extruder 0.0573
  MoveL (T18622) to (111.98, 103.84, 19.5) mm, rotated rx 180 ry 0 rz -180 deg; joints [1.326, 65.815, -27.764, 2.15, -38.07, -1.693]
  Call Extruder 0.01786
  MoveL (T18623) to (111.4, 103.84, 19.5) mm, rotated rx 180 ry 0 rz -180 deg; joints [1.323, 65.799, -27.735, 2.146, -38.083, -1.689]
  Call Extruder 0.0573
  MoveL (T18624) to (112.72, 105.16, 19.5) mm, rotated rx 180 ry 0 rz -180 deg; joints [1.323, 65.799, -27.735, 2.146, -38.083, -1.689]
  Call Extruder 0.01786
  MoveL (T18625) to (112.13, 105.16, 19.5) mm, rotated rx 180 ry 0 rz -180 deg; joints [1.323, 65.799, -27.735, 2.146, -38.083, -1.689]
  Call Extruder 0.0573
  MoveL (T18626) to (110.81, 103.84, 19.5) mm, rotated rx 180 ry 0 rz -180 deg; joints [1.323, 65.799, -27.735, 2.146, -38.083, -1.689]
  Call Extruder 0.01786
  MoveL (T18627) to (110.23, 103.84, 19.5) mm, rotated rx 180 ry 0 rz -180 deg; joints [1.321, 66.034, -28.177, 2.152, -37.877, -1.699]
  Call Extruder 0.0573
  MoveL (T18628) to (111.55, 105.16, 19.5) mm, rotated rx 180 ry 0 rz -180 deg; joints [1.321, 66.034, -28.177, 2.152, -37.877, -1.699]
  Call Extruder 0.01786
  MoveL (T18629) to (110.97, 105.16, 19.5) mm, rotated rx 180 ry 0 rz -180 deg; joints [1.321, 66.034, -28.177, 2.152, -37.877, -1.699]
  Call Extruder 0.0573
  MoveL (T18630) to (109.65, 103.84, 19.5) mm, rotated rx 180 ry 0 rz -180 deg; joints [1.321, 66.034, -28.177, 2.152, -37.877, -1.699]
  Call Extruder 0.01786
  MoveL (T18631) to (109.07, 103.84, 19.5) mm, rotated rx 180 ry 0 rz -180 deg; joints [1.321, 66.034, -28.177, 2.152, -37.877, -1.699]
  Call Extruder 0.0573
  MoveL (T18632) to (110.39, 105.16, 19.5) mm, rotated rx 180 ry 0 rz -180 deg; joints [1.321, 66.034, -28.177, 2.152, -37.877, -1.699]
  Call Extruder 0.01786
  MoveL (T18633) to (109.81, 105.16, 19.5) mm, rotated rx 180 ry 0 rz -180 deg; joints [1.707, 65.873, -28.281, 2.796, -37.625, -2.215]
  Call Extruder 0.0573
  MoveL (T18634) to (108.49, 103.84, 19.5) mm, rotated rx 180 ry 0 rz -180 deg; joints [1.707, 66.109, -28.317, 2.783, -37.825, -2.199]
  Call Extruder 0.01786
  MoveL (T18635) to (107.91, 103.84, 19.5) mm, rotated rx 180 ry 0 rz -180 deg; joints [1.707, 66.109, -28.317, 2.783, -37.825, -2.199]
  Call Extruder 0.0573
  MoveL (T18636) to (109.23, 105.16, 19.5) mm, rotated rx 180 ry 0 rz -180 deg; joints [1.707, 66.109, -28.317, 2.783, -37.825, -2.199]
  Call Extruder 0.01786
  MoveL (T18637) to (108.65, 105.16, 19.5) mm, rotated rx 180 ry 0 rz -180 deg; joints [1.707, 66.109, -28.317, 2.783, -37.825, -2.199]
  Call Extruder 0.0573
  MoveL (T18638) to (107.33, 103.84, 19.5) mm, rotated rx 180 ry 0 rz -180 deg; joints [1.707, 66.109, -28.317, 2.783, -37.825, -2.199]
  Call Extruder 0.01786
  MoveL (T18639) to (106.75, 103.84, 19.5) mm, rotated rx 180 ry 0 rz -180 deg; joints [1.707, 66.109, -28.317, 2.783, -37.825, -2.199]
  Call Extruder 0.0573
  MoveL (T18640) to (108.07, 105.16, 19.5) mm, rotated rx 180 ry 0 rz -180 deg; joints [1.707, 66.109, -28.317, 2.783, -37.825, -2.199]
  Call Extruder 0.01786
  MoveL (T18641) to (107.49, 105.16, 19.5) mm, rotated rx 180 ry 0 rz -180 deg; joints [1.707, 66.109, -28.317, 2.783, -37.825, -2.199]
  Call Extruder 0.0573
  MoveL (T18642) to (106.17, 103.84, 19.5) mm, rotated rx 180 ry 0 rz -180 deg; joints [1.707, 66.109, -28.317, 2.783, -37.825, -2.199]
  Call Extruder 0.01786
  MoveL (T18643) to (105.59, 103.84, 19.5) mm, rotated rx 180 ry 0 rz -180 deg; joints [1.442, 66.092, -28.284, 2.351, -37.831, -1.857]
  Call Extruder 0.08219
  MoveL (T18644) to (107.48, 105.73, 19.5) mm, rotated rx 180 ry 0 rz -180 deg; joints [1.442, 66.092, -28.284, 2.351, -37.831, -1.857]
  Call Extruder 0.01786
  MoveL (T18645) to (107.48, 106.32, 19.5) mm, rotated rx 180 ry 0 rz -180 deg; joints [1.657, 66.107, -28.313, 2.703, -37.825, -2.136]
  Call Extruder 0.10744
  MoveL (T18646) to (105.01, 103.84, 19.5) mm, rotated rx 180 ry 0 rz -180 deg; joints [1.657, 66.107, -28.313, 2.703, -37.825, -2.136]
  Call Extruder 0.01786
  MoveL (T18647) to (104.42, 103.84, 19.5) mm, rotated rx 180 ry 0 rz -180 deg; joints [1.679, 66.13, -28.355, 2.739, -37.806, -2.165]
  Call Extruder 0.1327
  MoveL (T18648) to (107.48, 106.9, 19.5) mm, rotated rx 180 ry 0 rz -180 deg; joints [1.679, 66.13, -28.355, 2.739, -37.806, -2.165]
  Call Extruder 0.01087
  MoveL (T18649) to (107.48, 107.25, 19.5) mm, rotated rx 180 ry 0 rz -180 deg; joints [1.679, 66.13, -28.355, 2.739, -37.806, -2.165]
  Call Extruder 0.01602
  MoveL (T18650) to (107.72, 107.72, 19.5) mm, rotated rx 180 ry 0 rz -180 deg; joints [1.679, 66.13, -28.355, 2.739, -37.806, -2.165]
  Call Extruder 0.16825
  MoveL (T18651) to (103.84, 103.84, 19.5) mm, rotated rx 180 ry 0 rz -180 deg; joints [1.679, 66.13, -28.355, 2.739, -37.806, -2.165]
  Call Extruder 0.01786
  MoveL (T18652) to (103.84, 104.42, 19.5) mm, rotated rx 180 ry 0 rz -180 deg; joints [1.743, 66.291, -28.659, 2.853, -37.667, -2.259]
  Call Extruder 0.19454
  MoveL (T18653) to (108.32, 108.9, 19.5) mm, rotated rx 180 ry 0 rz -180 deg; joints [1.743, 66.291, -28.659, 2.853, -37.667, -2.259]
  Call Extruder 0.04092
  MoveL (T18654) to (108.92, 110.09, 19.5) mm, rotated rx 180 ry 0 rz -180 deg; joints [1.743, 66.291, -28.659, 2.853, -37.667, -2.259]
  Call Extruder 0.22084
  MoveL (T18655) to (103.84, 105.01, 19.5) mm, rotated rx 180 ry 0 rz -180 deg; joints [1.821, 66.117, -28.332, 2.97, -37.822, -2.347]
  Call Extruder 0.01786
  MoveL (T18656) to (103.84, 105.59, 19.5) mm, rotated rx 180 ry 0 rz -180 deg; joints [1.821, 66.117, -28.332, 2.97, -37.822, -2.347]
  Call Extruder 0.24714
  MoveL (T18657) to (109.53, 111.27, 19.5) mm, rotated rx 180 ry 0 rz -180 deg; joints [1.821, 66.117, -28.332, 2.97, -37.822, -2.347]
  Call Extruder 0.04092
  MoveL (T18658) to (110.13, 112.46, 19.5) mm, rotated rx 180 ry 0 rz -180 deg; joints [1.941, 66.127, -28.35, 3.166, -37.819, -2.502]
  Call Extruder 0.27344
  MoveL (T18659) to (103.84, 106.17, 19.5) mm, rotated rx 180 ry 0 rz -180 deg; joints [1.941, 66.127, -28.35, 3.166, -37.819, -2.502]
  Call Extruder 0.01786
  MoveL (T18660) to (103.84, 106.75, 19.5) mm, rotated rx 180 ry 0 rz -180 deg; joints [3.239, 69.778, -35.207, 5.695, -34.704, -4.686]
  Call Extruder 0.29974
  MoveL (T18661) to (110.74, 113.64, 19.5) mm, rotated rx 180 ry 0 rz -180 deg; joints [3.239, 69.778, -35.207, 5.695, -34.704, -4.686]
  Call Extruder 0.04092
  MoveL (T18662) to (111.34, 114.83, 19.5) mm, rotated rx 180 ry 0 rz -180 deg; joints [3.239, 69.778, -35.207, 5.695, -34.704, -4.686]
  Call Extruder 0.32604
  MoveL (T18663) to (103.84, 107.33, 19.5) mm, rotated rx 180 ry 0 rz -180 deg; joints [3.239, 69.778, -35.207, 5.695, -34.704, -4.686]
  Call Extruder 0.01786
  MoveL (T18664) to (103.84, 107.91, 19.5) mm, rotated rx 180 ry 0 rz -180 deg; joints [3.232, 70.109, -35.829, 5.725, -34.414, -4.728]
  Call Extruder 0.34996
  MoveL (T18665) to (111.89, 115.96, 19.5) mm, rotated rx 180 ry 0 rz -180 deg; joints [3.232, 70.109, -35.829, 5.725, -34.414, -4.728]
  Call Extruder 0.01786
  MoveL (T18666) to (111.31, 115.96, 19.5) mm, rotated rx 180 ry 0 rz -180 deg; joints [3.232, 70.109, -35.829, 5.725, -34.414, -4.728]
  Call Extruder 0.32471
  MoveL (T18667) to (103.84, 108.49, 19.5) mm, rotated rx 180 ry 0 rz -180 deg; joints [2.845, 71.126, -37.739, 5.16, -33.494, -4.307]
  Call Extruder 0.01786
  MoveL (T18668) to (103.84, 109.07, 19.5) mm, rotated rx 180 ry 0 rz -180 deg; joints [2.845, 71.126, -37.739, 5.16, -33.494, -4.307]
  Call Extruder 0.29945
  MoveL (T18669) to (110.73, 115.96, 19.5) mm, rotated rx 180 ry 0 rz -180 deg; joints [3.211, 71.184, -37.848, 5.829, -33.473, -4.868]
  Call Extruder 0.01786
  MoveL (T18670) to (110.15, 115.96, 19.5) mm, rotated rx 180 ry 0 rz -180 deg; joints [3.211, 71.184, -37.848, 5.829, -33.473, -4.868]
  Call Extruder 0.2742
  MoveL (T18671) to (103.84, 109.65, 19.5) mm, rotated rx 180 ry 0 rz -180 deg; joints [3.211, 71.184, -37.848, 5.829, -33.473, -4.868]
  Call Extruder 0.01786
  MoveL (T18672) to (103.84, 110.23, 19.5) mm, rotated rx 180 ry 0 rz -180 deg; joints [1.893, 67.253, -30.464, 3.159, -36.831, -2.529]
  Call Extruder 0.24895
  MoveL (T18673) to (109.57, 115.96, 19.5) mm, rotated rx 180 ry 0 rz -180 deg; joints [1.893, 67.253, -30.464, 3.159, -36.831, -2.529]
  Call Extruder 0.01786
  MoveL (T18674) to (108.99, 115.96, 19.5) mm, rotated rx 180 ry 0 rz -180 deg; joints [1.895, 67.116, -30.207, 3.153, -36.951, -2.521]
  Call Extruder 0.22369
  MoveL (T18675) to (103.84, 110.82, 19.5) mm, rotated rx 180 ry 0 rz -180 deg; joints [1.895, 67.116, -30.207, 3.153, -36.951, -2.521]
  Call Extruder 0.01786
  MoveL (T18676) to (103.84, 111.4, 19.5) mm, rotated rx 180 ry 0 rz -180 deg; joints [1.895, 67.116, -30.207, 3.153, -36.951, -2.521]
  Call Extruder 0.19844
  MoveL (T18677) to (108.41, 115.96, 19.5) mm, rotated rx 180 ry 0 rz -180 deg; joints [2.319, 66.16, -28.412, 3.785, -37.808, -2.992]
  Call Extruder 0.01786
  MoveL (T18678) to (107.83, 115.96, 19.5) mm, rotated rx 180 ry 0 rz -180 deg; joints [2.319, 66.16, -28.412, 3.785, -37.808, -2.992]
  Call Extruder 0.17318
  MoveL (T18679) to (103.84, 111.98, 19.5) mm, rotated rx 180 ry 0 rz -180 deg; joints [2.319, 66.16, -28.412, 3.785, -37.808, -2.992]
  Call Extruder 0.01786
  MoveL (T18680) to (103.84, 112.56, 19.5) mm, rotated rx 180 ry 0 rz -180 deg; joints [2.44, 66.172, -28.435, 3.982, -37.804, -3.148]
  Call Extruder 0.1616
  MoveL (T18681) to (107.56, 116.28, 19.5) mm, rotated rx 180 ry 0 rz -180 deg; joints [2.44, 66.172, -28.435, 3.982, -37.804, -3.148]
  Call Extruder 0.01786
  MoveL (T18682) to (107.56, 116.86, 19.5) mm, rotated rx 180 ry 0 rz -180 deg; joints [3.266, 68.452, -32.716, 5.581, -35.865, -4.528]
  Call Extruder 0.1616
  MoveL (T18683) to (103.84, 113.14, 19.5) mm, rotated rx 180 ry 0 rz -180 deg; joints [3.266, 68.452, -32.716, 5.581, -35.865, -4.528]
  Call Extruder 0.01786
  MoveL (T18684) to (103.84, 113.72, 19.5) mm, rotated rx 180 ry 0 rz -180 deg; joints [3.26, 68.766, -33.305, 5.607, -35.591, -4.564]
  Call Extruder 0.1616
  MoveL (T18685) to (107.56, 117.44, 19.5) mm, rotated rx 180 ry 0 rz -180 deg; joints [3.26, 68.766, -33.305, 5.607, -35.591, -4.564]
  Call Extruder 0.01786
  MoveL (T18686) to (107.56, 118.02, 19.5) mm, rotated rx 180 ry 0 rz -180 deg; joints [2.685, 70.197, -35.994, 4.768, -34.296, -3.942]
  Call Extruder 0.1616
  MoveL (T18687) to (103.84, 114.3, 19.5) mm, rotated rx 180 ry 0 rz -180 deg; joints [2.685, 70.197, -35.994, 4.768, -34.296, -3.942]
  Call Extruder 0.01786
  MoveL (T18688) to (103.84, 114.88, 19.5) mm, rotated rx 180 ry 0 rz -180 deg; joints [2.754, 70.417, -36.407, 4.916, -34.108, -4.073]
  Call Extruder 0.1616
  MoveL (T18689) to (107.56, 118.6, 19.5) mm, rotated rx 180 ry 0 rz -180 deg; joints [2.754, 70.417, -36.407, 4.916, -34.108, -4.073]
  Call Extruder 0.01786
  MoveL (T18690) to (107.56, 119.18, 19.5) mm, rotated rx 180 ry 0 rz -180 deg; joints [2.754, 70.417, -36.407, 4.916, -34.108, -4.073]
  Call Extruder 0.16957
  MoveL (T18691) to (103.66, 115.28, 19.5) mm, rotated rx 180 ry 0 rz -180 deg; joints [2.754, 70.417, -36.407, 4.916, -34.108, -4.073]
  Set speed (45.0 mm/s)
  Call Extruder -1.6
  MoveL (T18692) to (103.66, 115.28, 19.5) mm, rotated rx 180 ry 0 rz -180 deg; joints [2.762, 70.48, -36.524, 4.936, -34.054, -4.093]
  Set speed (120.0 mm/s)
  MoveL (T18693) to (103.66, 115.28, 19.5) mm, rotated rx 180 ry 0 rz -180 deg; joints [2.762, 70.48, -36.524, 4.936, -34.054, -4.093]
  Call Extruder -0.38
  MoveL (T18694) to (104.42, 116.03, 19.5) mm, rotated rx 180 ry 0 rz -180 deg; joints [2.762, 70.48, -36.524, 4.936, -34.054, -4.093]
  Set speed (45.0 mm/s)
  Call Extruder -0.02
  MoveL (T18695) to (104.42, 116.03, 19.5) mm, rotated rx 180 ry 0 rz -180 deg; joints [2.762, 70.48, -36.524, 4.936, -34.054, -4.093]
  Set speed (150.0 mm/s)
  MoveL (T18696) to (104.42, 116.03, 21.5) mm, rotated rx 180 ry 0 rz -180 deg; joints [2.762, 70.48, -36.524, 4.936, -34.054, -4.093]
  MoveL (T18697) to (117.77, 105.57, 21.5) mm, rotated rx 180 ry 0 rz -180 deg; joints [2.756, 70.863, -37.245, 4.968, -33.718, -4.136]
  MoveL (T18698) to (117.77, 105.57, 19.5) mm, rotated rx 180 ry 0 rz -180 deg; joints [2.756, 70.863, -37.245, 4.968, -33.718, -4.136]
  Set speed (40.0 mm/s)
  Call Extruder 2.0
  MoveL (T18699) to (117.77, 105.57, 19.5) mm, rotated rx 180 ry 0 rz -180 deg; joints [2.756, 70.863, -37.245, 4.968, -33.718, -4.136]
  Call Extruder 0.14703
  MoveL (T18700) to (121.16, 108.96, 19.5) mm, rotated rx 180 ry 0 rz -180 deg; joints [2.756, 70.863, -37.245, 4.968, -33.718, -4.136]
  Call Extruder 0.01786
  MoveL (T18701) to (121.16, 109.54, 19.5) mm, rotated rx 180 ry 0 rz -180 deg; joints [2.756, 70.863, -37.245, 4.968, -33.718, -4.136]
  Call Extruder 0.13907
  MoveL (T18702) to (117.96, 106.34, 19.5) mm, rotated rx 180 ry 0 rz -180 deg; joints [2.756, 70.863, -37.245, 4.968, -33.718, -4.136]
  Call Extruder 0.01786
  MoveL (T18703) to (117.96, 106.92, 19.5) mm, rotated rx 180 ry 0 rz -180 deg; joints [2.756, 70.863, -37.245, 4.968, -33.718, -4.136]
  Call Extruder 0.13907
  MoveL (T18704) to (121.16, 110.12, 19.5) mm, rotated rx 180 ry 0 rz -180 deg; joints [2.761, 70.534, -36.627, 4.941, -34.006, -4.099]
  Call Extruder 0.01786
  MoveL (T18705) to (121.16, 110.7, 19.5) mm, rotated rx 180 ry 0 rz -180 deg; joints [2.761, 70.534, -36.627, 4.941, -34.006, -4.099]
  Call Extruder 0.13907
  MoveL (T18706) to (117.96, 107.5, 19.5) mm, rotated rx 180 ry 0 rz -180 deg; joints [2.761, 70.534, -36.627, 4.941, -34.006, -4.099]
  Call Extruder 0.01786
  MoveL (T18707) to (117.96, 108.08, 19.5) mm, rotated rx 180 ry 0 rz -180 deg; joints [2.761, 70.534, -36.627, 4.941, -34.006, -4.099]
  Call Extruder 0.13907
  MoveL (T18708) to (121.16, 111.28, 19.5) mm, rotated rx 180 ry 0 rz -180 deg; joints [2.761, 70.534, -36.627, 4.941, -34.006, -4.099]
  Call Extruder 0.01786
  MoveL (T18709) to (121.16, 111.86, 19.5) mm, rotated rx 180 ry 0 rz -180 deg; joints [2.761, 70.534, -36.627, 4.941, -34.006, -4.099]
  Call Extruder 0.13907
  MoveL (T18710) to (117.96, 108.66, 19.5) mm, rotated rx 180 ry 0 rz -180 deg; joints [2.761, 70.534, -36.627, 4.941, -34.006, -4.099]
  Call Extruder 0.01786
  MoveL (T18711) to (117.96, 109.24, 19.5) mm, rotated rx 180 ry 0 rz -180 deg; joints [2.761, 70.534, -36.627, 4.941, -34.006, -4.099]
  Call Extruder 0.13907
  MoveL (T18712) to (121.16, 112.44, 19.5) mm, rotated rx 180 ry 0 rz -180 deg; joints [2.761, 70.302, -36.586, 4.965, -33.816, -4.129]
  Call Extruder 0.01786
  MoveL (T18713) to (121.16, 113.02, 19.5) mm, rotated rx 180 ry 0 rz -180 deg; joints [1.813, 70.545, -37.042, 3.282, -33.546, -2.736]
  Call Extruder 0.15905
  MoveL (T18714) to (117.5, 109.36, 19.5) mm, rotated rx 180 ry 0 rz -180 deg; joints [1.813, 70.545, -37.042, 3.282, -33.546, -2.736]
  Call Extruder 0.01786
  MoveL (T18715) to (116.92, 109.36, 19.5) mm, rotated rx 180 ry 0 rz -180 deg; joints [1.813, 70.777, -37.083, 3.265, -33.737, -2.716]
  Call Extruder 0.1843
  MoveL (T18716) to (121.16, 113.6, 19.5) mm, rotated rx 180 ry 0 rz -180 deg; joints [1.813, 70.777, -37.083, 3.265, -33.737, -2.716]
  Call Extruder 0.01786
  MoveL (T18717) to (121.16, 114.19, 19.5) mm, rotated rx 180 ry 0 rz -180 deg; joints [1.813, 70.777, -37.083, 3.265, -33.737, -2.716]
  Call Extruder 0.20956
  MoveL (T18718) to (116.33, 109.36, 19.5) mm, rotated rx 180 ry 0 rz -180 deg; joints [1.813, 70.777, -37.083, 3.265, -33.737, -2.716]
  Call Extruder 0.01786
  MoveL (T18719) to (115.75, 109.36, 19.5) mm, rotated rx 180 ry 0 rz -180 deg; joints [1.813, 70.777, -37.083, 3.265, -33.737, -2.716]
  Call Extruder 0.23481
  MoveL (T18720) to (121.16, 114.77, 19.5) mm, rotated rx 180 ry 0 rz -180 deg; joints [1.813, 70.777, -37.083, 3.265, -33.737, -2.716]
  Call Extruder 0.01786
  MoveL (T18721) to (121.16, 115.35, 19.5) mm, rotated rx 180 ry 0 rz -180 deg; joints [1.813, 70.777, -37.083, 3.265, -33.737, -2.716]
  Call Extruder 0.26007
  MoveL (T18722) to (115.17, 109.36, 19.5) mm, rotated rx 180 ry 0 rz -180 deg; joints [1.813, 70.777, -37.083, 3.265, -33.737, -2.716]
  Call Extruder 0.01786
  MoveL (T18723) to (114.59, 109.36, 19.5) mm, rotated rx 180 ry 0 rz -180 deg; joints [1.813, 70.777, -37.083, 3.265, -33.737, -2.716]
  Call Extruder 0.28532
  MoveL (T18724) to (121.16, 115.93, 19.5) mm, rotated rx 180 ry 0 rz -180 deg; joints [1.813, 70.777, -37.083, 3.265, -33.737, -2.716]
  Call Extruder 0.01786
  MoveL (T18725) to (121.16, 116.51, 19.5) mm, rotated rx 180 ry 0 rz -180 deg; joints [1.886, 71.007, -37.516, 3.414, -33.538, -2.847]
  Call Extruder 0.31058
  MoveL (T18726) to (114.01, 109.36, 19.5) mm, rotated rx 180 ry 0 rz -180 deg; joints [1.946, 71.014, -37.527, 3.524, -33.536, -2.939]
  Call Extruder 0.01786
  MoveL (T18727) to (113.43, 109.36, 19.5) mm, rotated rx 180 ry 0 rz -180 deg; joints [1.946, 71.014, -37.527, 3.524, -33.536, -2.939]
  Call Extruder 0.33583
  MoveL (T18728) to (121.16, 117.09, 19.5) mm, rotated rx 180 ry 0 rz -180 deg; joints [1.946, 71.014, -37.527, 3.524, -33.536, -2.939]
  Call Extruder 0.01786
  MoveL (T18729) to (121.16, 117.67, 19.5) mm, rotated rx 180 ry 0 rz -180 deg; joints [1.946, 71.014, -37.527, 3.524, -33.536, -2.939]
  Call Extruder 0.31968
  MoveL (T18730) to (113.8, 110.32, 19.5) mm, rotated rx 180 ry 0 rz -180 deg; joints [1.833, 70.657, -36.857, 3.293, -33.844, -2.736]
  Call Extruder 0.04109
  MoveL (T18731) to (114.41, 111.51, 19.5) mm, rotated rx 180 ry 0 rz -180 deg; joints [1.833, 70.657, -36.857, 3.293, -33.844, -2.736]
  Call Extruder 0.29321
  MoveL (T18732) to (121.16, 118.25, 19.5) mm, rotated rx 180 ry 0 rz -180 deg; joints [1.835, 70.479, -36.523, 3.283, -34, -2.723]
  Call Extruder 0.01786
  MoveL (T18733) to (121.16, 118.83, 19.5) mm, rotated rx 180 ry 0 rz -180 deg; joints [1.835, 70.479, -36.523, 3.283, -34, -2.723]
  Call Extruder 0.26675
  MoveL (T18734) to (115.02, 112.7, 19.5) mm, rotated rx 180 ry 0 rz -180 deg; joints [1.835, 70.479, -36.523, 3.283, -34, -2.723]
  Call Extruder 0.04109
  MoveL (T18735) to (115.63, 113.89, 19.5) mm, rotated rx 180 ry 0 rz -180 deg; joints [2.007, 71.02, -37.539, 3.635, -33.534, -3.031]
  Call Extruder 0.24028
  MoveL (T18736) to (121.16, 119.41, 19.5) mm, rotated rx 180 ry 0 rz -180 deg; joints [2.007, 71.02, -37.539, 3.635, -33.534, -3.031]
  Call Extruder 0.01786
  MoveL (T18737) to (121.16, 119.99, 19.5) mm, rotated rx 180 ry 0 rz -180 deg; joints [2.068, 71.026, -37.551, 3.745, -33.531, -3.123]
  Call Extruder 0.21381
  MoveL (T18738) to (116.24, 115.08, 19.5) mm, rotated rx 180 ry 0 rz -180 deg; joints [2.068, 71.026, -37.551, 3.745, -33.531, -3.123]
  Call Extruder 0.04109
  MoveL (T18739) to (116.85, 116.27, 19.5) mm, rotated rx 180 ry 0 rz -180 deg; joints [1.852, 70.347, -36.275, 3.303, -34.116, -2.735]
  Call Extruder 0.18734
  MoveL (T18740) to (121.16, 120.58, 19.5) mm, rotated rx 180 ry 0 rz -180 deg; joints [1.852, 70.347, -36.275, 3.303, -34.116, -2.735]
  Call Extruder 0.01786
  MoveL (T18741) to (121.16, 121.16, 19.5) mm, rotated rx 180 ry 0 rz -180 deg; joints [1.883, 70.262, -36.116, 3.352, -34.192, -2.774]
  Call Extruder 0.16087
  MoveL (T18742) to (117.45, 117.45, 19.5) mm, rotated rx 180 ry 0 rz -180 deg; joints [1.883, 70.262, -36.116, 3.352, -34.192, -2.774]
  Call Extruder 0.02137
  MoveL (T18743) to (117.77, 118.07, 19.5) mm, rotated rx 180 ry 0 rz -180 deg; joints [1.883, 70.262, -36.116, 3.352, -34.192, -2.774]
  Call Extruder 0.00857
  MoveL (T18744) to (117.77, 118.35, 19.5) mm, rotated rx 180 ry 0 rz -180 deg; joints [2.129, 71.033, -37.564, 3.856, -33.529, -3.215]
  Call Extruder 0.12185
  MoveL (T18745) to (120.58, 121.16, 19.5) mm, rotated rx 180 ry 0 rz -180 deg; joints [2.129, 71.033, -37.564, 3.856, -33.529, -3.215]
  Call Extruder 0.01786
  MoveL (T18746) to (119.99, 121.16, 19.5) mm, rotated rx 180 ry 0 rz -180 deg; joints [2.129, 71.033, -37.564, 3.856, -33.529, -3.215]
  Call Extruder 0.09659
  MoveL (T18747) to (117.77, 118.93, 19.5) mm, rotated rx 180 ry 0 rz -180 deg; joints [2.189, 71.04, -37.576, 3.966, -33.526, -3.308]
  Call Extruder 0.01786
  MoveL (T18748) to (117.77, 119.52, 19.5) mm, rotated rx 180 ry 0 rz -180 deg; joints [2.189, 71.04, -37.576, 3.966, -33.526, -3.308]
  Call Extruder 0.07134
  MoveL (T18749) to (119.41, 121.16, 19.5) mm, rotated rx 180 ry 0 rz -180 deg; joints [1.915, 70.177, -35.957, 3.402, -34.268, -2.812]
  Call Extruder 0.01786
  MoveL (T18750) to (118.83, 121.16, 19.5) mm, rotated rx 180 ry 0 rz -180 deg; joints [1.915, 70.177, -35.957, 3.402, -34.268, -2.812]
  Call Extruder 0.04608
  MoveL (T18751) to (117.77, 120.1, 19.5) mm, rotated rx 180 ry 0 rz -180 deg; joints [1.915, 70.177, -35.957, 3.402, -34.268, -2.812]
  Call Extruder 0.00206
  MoveL (T18752) to (117.77, 120.16, 19.5) mm, rotated rx 180 ry 0 rz -180 deg; joints [1.946, 70.093, -35.798, 3.451, -34.343, -2.851]
  Call Extruder 0.0158
  MoveL (T18753) to (117.26, 120.16, 19.5) mm, rotated rx 180 ry 0 rz -180 deg; joints [1.946, 70.093, -35.798, 3.451, -34.343, -2.851]
  Call Extruder 0.04317
  MoveL (T18754) to (118.25, 121.16, 19.5) mm, rotated rx 180 ry 0 rz -180 deg; joints [1.946, 70.093, -35.798, 3.451, -34.343, -2.851]
  Call Extruder 0.01786
  MoveL (T18755) to (117.67, 121.16, 19.5) mm, rotated rx 180 ry 0 rz -180 deg; joints [1.946, 70.093, -35.798, 3.451, -34.343, -2.851]
  Call Extruder 0.04317
  MoveL (T18756) to (116.68, 120.16, 19.5) mm, rotated rx 180 ry 0 rz -180 deg; joints [2.25, 71.047, -37.59, 4.076, -33.524, -3.4]
  Call Extruder 0.01786
  MoveL (T18757) to (116.1, 120.16, 19.5) mm, rotated rx 180 ry 0 rz -180 deg; joints [2.25, 71.047, -37.59, 4.076, -33.524, -3.4]
  Call Extruder 0.04317
  MoveL (T18758) to (117.09, 121.16, 19.5) mm, rotated rx 180 ry 0 rz -180 deg; joints [2.25, 71.047, -37.59, 4.076, -33.524, -3.4]
  Call Extruder 0.01786
  MoveL (T18759) to (116.51, 121.16, 19.5) mm, rotated rx 180 ry 0 rz -180 deg; joints [2.25, 71.047, -37.59, 4.076, -33.524, -3.4]
  Call Extruder 0.04317
  MoveL (T18760) to (115.52, 120.16, 19.5) mm, rotated rx 180 ry 0 rz -180 deg; joints [2.311, 71.054, -37.603, 4.187, -33.521, -3.492]
  Call Extruder 0.01786
  MoveL (T18761) to (114.93, 120.16, 19.5) mm, rotated rx 180 ry 0 rz -180 deg; joints [2.311, 71.054, -37.603, 4.187, -33.521, -3.492]
  Call Extruder 0.04317
  MoveL (T18762) to (115.93, 121.16, 19.5) mm, rotated rx 180 ry 0 rz -180 deg; joints [2.311, 71.054, -37.603, 4.187, -33.521, -3.492]
  Call Extruder 0.01786
  MoveL (T18763) to (115.35, 121.16, 19.5) mm, rotated rx 180 ry 0 rz -180 deg; joints [2.311, 71.054, -37.603, 4.187, -33.521, -3.492]
  Call Extruder 0.04317
  MoveL (T18764) to (114.35, 120.16, 19.5) mm, rotated rx 180 ry 0 rz -180 deg; joints [1.978, 70.009, -35.641, 3.5, -34.418, -2.889]
  Call Extruder 0.01786
  MoveL (T18765) to (113.77, 120.16, 19.5) mm, rotated rx 180 ry 0 rz -180 deg; joints [1.978, 70.009, -35.641, 3.5, -34.418, -2.889]
  Call Extruder 0.04317
  MoveL (T18766) to (114.77, 121.16, 19.5) mm, rotated rx 180 ry 0 rz -180 deg; joints [1.978, 70.009, -35.641, 3.5, -34.418, -2.889]
  Call Extruder 0.01786
  MoveL (T18767) to (114.18, 121.16, 19.5) mm, rotated rx 180 ry 0 rz -180 deg; joints [2.009, 69.926, -35.484, 3.55, -34.493, -2.927]
  Call Extruder 0.04317
  MoveL (T18768) to (113.19, 120.16, 19.5) mm, rotated rx 180 ry 0 rz -180 deg; joints [2.009, 69.926, -35.484, 3.55, -34.493, -2.927]
  Call Extruder 0.01786
  MoveL (T18769) to (112.61, 120.16, 19.5) mm, rotated rx 180 ry 0 rz -180 deg; joints [2.371, 71.061, -37.617, 4.297, -33.518, -3.585]
  Call Extruder 0.04317
  MoveL (T18770) to (113.6, 121.16, 19.5) mm, rotated rx 180 ry 0 rz -180 deg; joints [2.371, 71.061, -37.617, 4.297, -33.518, -3.585]
  Call Extruder 0.01786
  MoveL (T18771) to (113.02, 121.16, 19.5) mm, rotated rx 180 ry 0 rz -180 deg; joints [2.371, 71.061, -37.617, 4.297, -33.518, -3.585]
  Call Extruder 0.04317
  MoveL (T18772) to (112.03, 120.16, 19.5) mm, rotated rx 180 ry 0 rz -180 deg; joints [2.432, 71.069, -37.631, 4.408, -33.516, -3.677]
  Call Extruder 0.01786
  MoveL (T18773) to (111.45, 120.16, 19.5) mm, rotated rx 180 ry 0 rz -180 deg; joints [2.432, 71.069, -37.631, 4.408, -33.516, -3.677]
  Call Extruder 0.04317
  MoveL (T18774) to (112.44, 121.16, 19.5) mm, rotated rx 180 ry 0 rz -180 deg; joints [2.432, 71.069, -37.631, 4.408, -33.516, -3.677]
  Call Extruder 0.01786
  MoveL (T18775) to (111.86, 121.16, 19.5) mm, rotated rx 180 ry 0 rz -180 deg; joints [2.041, 69.843, -35.328, 3.599, -34.568, -2.965]
  Call Extruder 0.04317
  MoveL (T18776) to (110.87, 120.16, 19.5) mm, rotated rx 180 ry 0 rz -180 deg; joints [2.041, 69.843, -35.328, 3.599, -34.568, -2.965]
  Call Extruder 0.01786
  MoveL (T18777) to (110.29, 120.16, 19.5) mm, rotated rx 180 ry 0 rz -180 deg; joints [2.041, 69.843, -35.328, 3.599, -34.568, -2.965]
  Call Extruder 0.04317
  MoveL (T18778) to (111.28, 121.16, 19.5) mm, rotated rx 180 ry 0 rz -180 deg; joints [2.048, 69.824, -35.293, 3.61, -34.584, -2.973]
  Call Extruder 0.01786
  MoveL (T18779) to (110.7, 121.16, 19.5) mm, rotated rx 180 ry 0 rz -180 deg; joints [2.048, 69.824, -35.293, 3.61, -34.584, -2.973]
  Call Extruder 0.04317
  MoveL (T18780) to (109.71, 120.16, 19.5) mm, rotated rx 180 ry 0 rz -180 deg; joints [2.048, 69.824, -35.293, 3.61, -34.584, -2.973]
  Call Extruder 0.01786
  MoveL (T18781) to (109.12, 120.16, 19.5) mm, rotated rx 180 ry 0 rz -180 deg; joints [2.048, 69.824, -35.293, 3.61, -34.584, -2.973]
  Call Extruder 0.04317
  MoveL (T18782) to (110.12, 121.16, 19.5) mm, rotated rx 180 ry 0 rz -180 deg; joints [2.048, 69.824, -35.293, 3.61, -34.584, -2.973]
  Call Extruder 0.01786
  MoveL (T18783) to (109.54, 121.16, 19.5) mm, rotated rx 180 ry 0 rz -180 deg; joints [2.053, 69.819, -35.282, 3.619, -34.59, -2.98]
  Call Extruder 0.05113
  MoveL (T18784) to (108.36, 119.98, 19.5) mm, rotated rx 180 ry 0 rz -180 deg; joints [2.053, 69.819, -35.282, 3.619, -34.59, -2.98]
  Set speed (150.0 mm/s)
  MoveL (T18785) to (109.14, 121.34, 19.5) mm, rotated rx 180 ry 0 rz -180 deg; joints [2.053, 69.819, -35.282, 3.619, -34.59, -2.98]
  Set speed (40.0 mm/s)
  MoveL (T18786) to (109.14, 121.34, 19.5) mm, rotated rx 180 ry 0 rz -180 deg; joints [2.053, 69.819, -35.282, 3.619, -34.59, -2.98]
  Call Extruder 0.05113
  MoveL (T18787) to (107.96, 120.16, 19.5) mm, rotated rx 180 ry 0 rz -180 deg; joints [2.093, 69.823, -35.29, 3.689, -34.588, -3.039]
  Call Extruder 0.01234
  MoveL (T18788) to (107.56, 120.16, 19.5) mm, rotated rx 180 ry 0 rz -180 deg; joints [2.093, 69.823, -35.29, 3.689, -34.588, -3.039]
  Call Extruder 0.01234
  MoveL (T18789) to (107.56, 119.76, 19.5) mm, rotated rx 180 ry 0 rz -180 deg; joints [2.493, 71.077, -37.646, 4.518, -33.513, -3.769]
  Call Extruder 0.1616
  MoveL (T18790) to (103.84, 116.04, 19.5) mm, rotated rx 180 ry 0 rz -180 deg; joints [2.493, 71.077, -37.646, 4.518, -33.513, -3.769]
  Call Extruder 0.01786
  MoveL (T18791) to (103.84, 116.62, 19.5) mm, rotated rx 180 ry 0 rz -180 deg; joints [2.553, 71.085, -37.661, 4.629, -33.51, -3.862]
  Call Extruder 0.19697
  MoveL (T18792) to (108.38, 121.16, 19.5) mm, rotated rx 180 ry 0 rz -180 deg; joints [2.553, 71.085, -37.661, 4.629, -33.51, -3.862]
  Call Extruder 0.01786
  MoveL (T18793) to (107.79, 121.16, 19.5) mm, rotated rx 180 ry 0 rz -180 deg; joints [2.553, 71.085, -37.661, 4.629, -33.51, -3.862]
  Call Extruder 0.17171
  MoveL (T18794) to (103.84, 117.21, 19.5) mm, rotated rx 180 ry 0 rz -180 deg; joints [2.154, 69.829, -35.302, 3.797, -34.586, -3.128]
  Call Extruder 0.01786
  MoveL (T18795) to (103.84, 117.79, 19.5) mm, rotated rx 180 ry 0 rz -180 deg; joints [2.154, 69.829, -35.302, 3.797, -34.586, -3.128]
  Call Extruder 0.14646
  MoveL (T18796) to (107.21, 121.16, 19.5) mm, rotated rx 180 ry 0 rz -180 deg; joints [2.154, 69.829, -35.302, 3.797, -34.586, -3.128]
  Call Extruder 0.01786
  MoveL (T18797) to (106.63, 121.16, 19.5) mm, rotated rx 180 ry 0 rz -180 deg; joints [2.216, 69.835, -35.314, 3.906, -34.584, -3.217]
  Call Extruder 0.1212
  MoveL (T18798) to (103.84, 118.37, 19.5) mm, rotated rx 180 ry 0 rz -180 deg; joints [2.216, 69.835, -35.314, 3.906, -34.584, -3.217]
  Call Extruder 0.01786
  MoveL (T18799) to (103.84, 118.95, 19.5) mm, rotated rx 180 ry 0 rz -180 deg; joints [2.216, 69.835, -35.314, 3.906, -34.584, -3.217]
  Call Extruder 0.09595
  MoveL (T18800) to (106.05, 121.16, 19.5) mm, rotated rx 180 ry 0 rz -180 deg; joints [2.614, 71.093, -37.677, 4.739, -33.507, -3.954]
  Call Extruder 0.01786
  MoveL (T18801) to (105.47, 121.16, 19.5) mm, rotated rx 180 ry 0 rz -180 deg; joints [2.614, 71.093, -37.677, 4.739, -33.507, -3.954]
  Call Extruder 0.07069
  MoveL (T18802) to (103.84, 119.53, 19.5) mm, rotated rx 180 ry 0 rz -180 deg; joints [2.675, 71.101, -37.692, 4.85, -33.504, -4.047]
  Call Extruder 0.01786
  MoveL (T18803) to (103.84, 120.11, 19.5) mm, rotated rx 180 ry 0 rz -180 deg; joints [2.675, 71.101, -37.692, 4.85, -33.504, -4.047]
  Call Extruder 0.04544
  MoveL (T18804) to (104.89, 121.16, 19.5) mm, rotated rx 180 ry 0 rz -180 deg; joints [2.277, 69.842, -35.326, 4.014, -34.581, -3.306]
  Call Extruder 0.01786
  MoveL (T18805) to (104.31, 121.16, 19.5) mm, rotated rx 180 ry 0 rz -180 deg; joints [2.338, 69.849, -35.339, 4.122, -34.579, -3.395]
  Call Extruder 0.02815
  MoveL (T18806) to (103.66, 120.51, 19.5) mm, rotated rx 180 ry 0 rz -180 deg; joints [2.338, 69.849, -35.339, 4.122, -34.579, -3.395]
  Set speed (45.0 mm/s)
  Call Extruder -1.6
  MoveL (T18807) to (103.66, 120.51, 19.5) mm, rotated rx 180 ry 0 rz -180 deg; joints [2.71, 71.027, -37.552, 4.905, -33.571, -4.09]
  Set speed (120.0 mm/s)
  MoveL (T18808) to (103.66, 120.51, 19.5) mm, rotated rx 180 ry 0 rz -180 deg; joints [2.71, 71.027, -37.552, 4.905, -33.571, -4.09]
  Call Extruder -0.3262
  MoveL (T18809) to (104.31, 121.16, 19.5) mm, rotated rx 180 ry 0 rz -180 deg; joints [2.713, 70.846, -37.213, 4.89, -33.73, -4.07]
  Call Extruder -0.0538
  MoveL (T18810) to (104.46, 121.16, 19.5) mm, rotated rx 180 ry 0 rz -180 deg; joints [2.713, 70.846, -37.213, 4.89, -33.73, -4.07]
  Set speed (45.0 mm/s)
  Call Extruder -0.02
  MoveL (T18811) to (104.46, 121.16, 19.5) mm, rotated rx 180 ry 0 rz -180 deg; joints [2.399, 69.856, -35.353, 4.23, -34.576, -3.485]
  Set speed (150.0 mm/s)
  MoveL (T18812) to (104.46, 121.16, 21.5) mm, rotated rx 180 ry 0 rz -180 deg; joints [2.399, 69.856, -35.353, 4.23, -34.576, -3.485]
  MoveL (T18813) to (109.4, 105.47, 21.5) mm, rotated rx 180 ry 0 rz -180 deg; joints [2.399, 69.856, -35.353, 4.23, -34.576, -3.485]
  MoveL (T18814) to (109.4, 105.47, 19.7) mm, rotated rx 180 ry 0 rz -180 deg; joints [2.46, 69.863, -35.366, 4.338, -34.574, -3.574]
  Set speed (40.0 mm/s)
  Call Extruder 2.0
  MoveL (T18815) to (109.4, 105.47, 19.7) mm, rotated rx 180 ry 0 rz -180 deg; joints [2.46, 69.863, -35.366, 4.338, -34.574, -3.574]
  Call Extruder 0.25145
  MoveL (T18816) to (117.65, 105.47, 19.7) mm, rotated rx 180 ry 0 rz -180 deg; joints [2.716, 70.667, -36.877, 4.875, -33.886, -4.05]
  Call Extruder 0.10939
  MoveL (T18817) to (117.65, 109.06, 19.7) mm, rotated rx 180 ry 0 rz -180 deg; joints [2.716, 70.667, -36.877, 4.875, -33.886, -4.05]
  Call Extruder 0.14732
  MoveL (T18818) to (112.81, 109.06, 19.7) mm, rotated rx 180 ry 0 rz -180 deg; joints [2.716, 70.667, -36.877, 4.875, -33.886, -4.05]
  Call Extruder 0.31102
  MoveL (T18819) to (117.47, 118.15, 19.7) mm, rotated rx 180 ry 0 rz -180 deg; joints [2.719, 70.498, -36.559, 4.861, -34.035, -4.032]
  Call Extruder 0.05209
  MoveL (T18820) to (117.47, 119.86, 19.7) mm, rotated rx 180 ry 0 rz -180 deg; joints [2.719, 70.498, -36.559, 4.861, -34.035, -4.032]
  Call Extruder 0.29244
  MoveL (T18821) to (107.87, 119.86, 19.7) mm, rotated rx 180 ry 0 rz -180 deg; joints [2.719, 70.498, -36.559, 4.861, -34.035, -4.032]
  Call Extruder 0.10939
  MoveL (T18822) to (107.87, 116.27, 19.7) mm, rotated rx 180 ry 0 rz -180 deg; joints [2.717, 70.483, -36.531, 4.856, -34.048, -4.027]
  Call Extruder 0.13869
  MoveL (T18823) to (112.42, 116.27, 19.7) mm, rotated rx 180 ry 0 rz -180 deg; joints [2.503, 69.814, -35.273, 4.408, -34.62, -3.63]
  Call Extruder 0.31084
  MoveL (T18824) to (107.78, 107.18, 19.7) mm, rotated rx 180 ry 0 rz -180 deg; joints [2.503, 69.814, -35.273, 4.408, -34.62, -3.63]
  Call Extruder 0.05206
  MoveL (T18825) to (107.78, 105.47, 19.7) mm, rotated rx 180 ry 0 rz -180 deg; joints [2.503, 69.814, -35.273, 4.408, -34.62, -3.63]
  Call Extruder 0.04735
  MoveL (T18826) to (109.34, 105.47, 19.7) mm, rotated rx 180 ry 0 rz -180 deg; joints [2.503, 69.814, -35.273, 4.408, -34.62, -3.63]
  Set speed (150.0 mm/s)
  MoveL (T18827) to (109, 105.88, 19.7) mm, rotated rx 180 ry 0 rz -180 deg; joints [2.503, 69.814, -35.273, 4.408, -34.62, -3.63]
  Set speed (40.0 mm/s)
  MoveL (T18828) to (109, 105.88, 19.7) mm, rotated rx 180 ry 0 rz -180 deg; joints [2.503, 69.814, -35.273, 4.408, -34.62, -3.63]
  Call Extruder 0.25124
  MoveL (T18829) to (117.24, 105.88, 19.7) mm, rotated rx 180 ry 0 rz -180 deg; joints [2.503, 69.814, -35.273, 4.408, -34.62, -3.63]
  Call Extruder 0.08459
  MoveL (T18830) to (117.24, 108.65, 19.7) mm, rotated rx 180 ry 0 rz -180 deg; joints [2.503, 69.814, -35.273, 4.408, -34.62, -3.63]
  Call Extruder 0.1552
  MoveL (T18831) to (112.15, 108.65, 19.7) mm, rotated rx 180 ry 0 rz -180 deg; joints [2.503, 69.814, -35.273, 4.408, -34.62, -3.63]
  Call Extruder 0.32831
  MoveL (T18832) to (117.06, 118.25, 19.7) mm, rotated rx 180 ry 0 rz -180 deg; joints [2.503, 69.814, -35.273, 4.408, -34.62, -3.63]
  Call Extruder 0.0367
  MoveL (T18833) to (117.06, 119.45, 19.7) mm, rotated rx 180 ry 0 rz -180 deg; joints [2.503, 69.814, -35.273, 4.408, -34.62, -3.63]
  Call Extruder 0.26763
  MoveL (T18834) to (108.27, 119.45, 19.7) mm, rotated rx 180 ry 0 rz -180 deg; joints [2.503, 69.814, -35.273, 4.408, -34.62, -3.63]
  Call Extruder 0.08459
  MoveL (T18835) to (108.27, 116.67, 19.7) mm, rotated rx 180 ry 0 rz -180 deg; joints [2.579, 70.049, -35.714, 4.566, -34.419, -3.769]
  Call Extruder 0.14654
  MoveL (T18836) to (113.08, 116.67, 19.7) mm, rotated rx 180 ry 0 rz -180 deg; joints [2.579, 70.049, -35.714, 4.566, -34.419, -3.769]
  Call Extruder 0.32811
  MoveL (T18837) to (108.19, 107.08, 19.7) mm, rotated rx 180 ry 0 rz -180 deg; joints [2.579, 70.049, -35.714, 4.566, -34.419, -3.769]
  Call Extruder 0.03668
  MoveL (T18838) to (108.19, 105.88, 19.7) mm, rotated rx 180 ry 0 rz -180 deg; joints [2.579, 70.049, -35.714, 4.566, -34.419, -3.769]
  Call Extruder 0.02276
  MoveL (T18839) to (108.94, 105.88, 19.7) mm, rotated rx 180 ry 0 rz -180 deg; joints [2.579, 70.049, -35.714, 4.566, -34.419, -3.769]
  Set speed (150.0 mm/s)
  MoveL (T18840) to (108.6, 106.28, 19.7) mm, rotated rx 180 ry 0 rz -180 deg; joints [2.579, 70.049, -35.714, 4.566, -34.419, -3.769]
  Set speed (25.0 mm/s)
  MoveL (T18841) to (108.6, 106.28, 19.7) mm, rotated rx 180 ry 0 rz -180 deg; joints [1.869, 68.935, -34.022, 3.263, -34.957, -2.675]
  Call Extruder 0.25102
  MoveL (T18842) to (116.84, 106.28, 19.7) mm, rotated rx 180 ry 0 rz -180 deg; joints [1.869, 69.168, -34.061, 3.247, -35.151, -2.656]
  Call Extruder 0.05979
  MoveL (T18843) to (116.84, 108.25, 19.7) mm, rotated rx 180 ry 0 rz -180 deg; joints [1.869, 69.168, -34.061, 3.247, -35.151, -2.656]
  Call Extruder 0.16307
  MoveL (T18844) to (111.48, 108.25, 19.7) mm, rotated rx 180 ry 0 rz -180 deg; joints [1.869, 69.168, -34.061, 3.247, -35.151, -2.656]
  Call Extruder 0.3456
  MoveL (T18845) to (116.65, 118.34, 19.7) mm, rotated rx 180 ry 0 rz -180 deg; joints [1.869, 69.168, -34.061, 3.247, -35.151, -2.656]
  Call Extruder 0.02131
  MoveL (T18846) to (116.65, 119.04, 19.7) mm, rotated rx 180 ry 0 rz -180 deg; joints [1.869, 69.168, -34.061, 3.247, -35.151, -2.656]
  Call Extruder 0.24283
  MoveL (T18847) to (108.68, 119.04, 19.7) mm, rotated rx 180 ry 0 rz -180 deg; joints [1.869, 69.168, -34.061, 3.247, -35.151, -2.656]
  Call Extruder 0.05979
  MoveL (T18848) to (108.68, 117.08, 19.7) mm, rotated rx 180 ry 0 rz -180 deg; joints [1.869, 69.168, -34.061, 3.247, -35.151, -2.656]
  Call Extruder 0.15438
